KUKA KRL program: EPS_2_251491_MH03_A_20251118025954.src

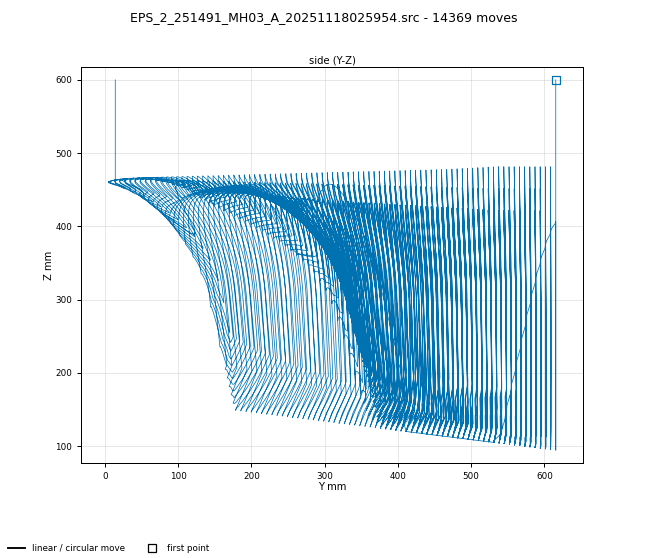
[picture p0: tool path of EPS_2_251491_MH03_A_20251118025954.src, 14369 of 14371 moves have a stored position in this frame; points joined in program order, loops and branches not executed]
&ACCESS RVP
&REL 4
&COMMENT QRS 19112012
&PARAM EDITMASK = *
DEF PART()
EXT BAS (BAS_COMMAND :IN,REAL :IN )
INT I
BAS (#INITMOV,0 )

;KUKA QRS Post kuka4.cps  Date:22-06-2017 !

File_ID=2921

QRS_PRE_INIT()

;Init var - Until changes are made in qrs_pre_init
Outlet_Square_prg=0
Inlet_1_Square_prg=0
Inlet_2_Square_prg=0
Inlet_3_Square_prg=0
Inlet_4_Square_prg=0
Inlet_5_Square_prg=0

Outlet_1={X 0.000, Y 534.640, Z 332.000, B 0.000, E1 0.000 }
Inlet_1={X 0.000, Y 539.010, Z 272.000, B 0.000, E1 90.000 }
Inlet_2={X 0.000, Y 536.830, Z 302.000, B 0.000, E1 207.000 }
Inlet_3={X 0.000, Y 539.010, Z 272.000, B 0.000, E1 270.000 }
Outlet_1_type=299
Inlet_1_type=299
Inlet_2_type=299
Inlet_3_type=299
;QRS#1=Sidecore dimensions
;QRS#2=300-12" PVC SDR 35
;QRS#3=300-12" PVC SDR 35
;QRS#4=300-12" PVC SDR 35
;QRS#5=300-12" PVC SDR 35
;QRS#6=
;QRS#7=
;QRS#8=
;QRS#9=16M PSX
;QRS#10=16M PSX
;QRS#11=16M PSX
;QRS#12=16M PSX
;QRS#13=
;QRS#14=
;QRS#15=
;QRS#16=1220x127x762 2,5'
;QRS#17=EPS Height
;QRS#18=481,5
;QRS#19=*
;QRS#20= UPDATED VERSION 22-06-2017
;QRS#21=*
Outlet_Square=0150
Inlet_1_Square=0150
Inlet_2_Square=0150
Inlet_3_Square=0150
Inlet_4_Square=0
Inlet_5_Square=0
Mill_Square=1
Outlet_Square_Prg=206
Inlet_1_Square_prg=206
Inlet_2_Square_prg=206
Inlet_3_Square_prg=206

QRS_INIT()

$ADVANCE=5

; T1
PTP {E1 173.529,E2 173.529}
PTP {X 0,Y 615.494,A -85,B 0,C 180,E1 173.529,E2 173.529,E3 0,E4 0,E5 0,E6 0}
QRS_SPEED_INIT()
LIN {X 0,Y 615.494,Z 600,A -85,B 0,C 180,E1 173.529,E2 173.529,E3 0,E4 0,E5 0,E6 0} C_VEL
LIN {X 0,Y 615.494,Z 417.846,A -85,B 0,C 180,E1 173.529,E2 173.529} C_VEL
LIN {X 0,Y 615.494,Z 408.199,A -85,B 0,C 180,E1 173.529,E2 173.529} C_VEL
LIN {X 0,Y 615.491,Z 406.378,A -85,B 0,C 180,E1 173.42,E2 173.42} C_VEL
LIN {X 0,Y 615.494,Z 399.659,A -85,B 0,C 180,E1 172.124,E2 172.124} C_VEL
LIN {X 0,Y 615.491,Z 391.142,A -85,B 0,C 180,E1 170.801,E2 170.801} C_VEL
LIN {X 0,Y 615.494,Z 382.064,A -85,B 0,C 180,E1 169.639,E2 169.639} C_VEL
LIN {X 0,Y 615.493,Z 372.79,A -85,B 0,C 180,E1 168.64,E2 168.64} C_VEL
LIN {X 0,Y 615.496,Z 360.819,A -85,B 0,C 180,E1 167.554,E2 167.554} C_VEL
LIN {X 0,Y 615.497,Z 348.577,A -85,B 0,C 180,E1 166.631,E2 166.631} C_VEL
LIN {X 0,Y 615.496,Z 335.878,A -85,B 0,C 180,E1 165.834,E2 165.834} C_VEL
LIN {X 0,Y 615.481,Z 321.775,A -85,B 0,C 180,E1 165.112,E2 165.112} C_VEL
LIN {X 0,Y 615.491,Z 307.115,A -85,B 0,C 180,E1 164.519,E2 164.519} C_VEL
LIN {X 0,Y 615.495,Z 292.173,A -85,B 0,C 180,E1 164.062,E2 164.062} C_VEL
LIN {X 0,Y 615.483,Z 277.013,A -85,B 0,C 180,E1 163.738,E2 163.738} C_VEL
LIN {X 0,Y 615.449,Z 230.182,A -85,B 0,C 180,E1 163.156,E2 163.156} C_VEL
LIN {X 0,Y 615.473,Z 111.41,A -85,B 0,C 180,E1 161.725,E2 161.725} C_VEL
LIN {X 0,Y 615.445,Z 94.319,A -85,B 0,C 180,E1 159.337,E2 159.337} C_VEL
LIN {X 0,Y 615.446,Z 94.317,A -85,B 0,C 180,E1 157.154,E2 157.154} C_VEL
LIN {X 0,Y 615.497,Z 94.322,A -85,B 0,C 180,E1 154.284,E2 154.284} C_VEL
LIN {X 0,Y 615.441,Z 94.32,A -85,B 0,C 180,E1 151.558,E2 151.558} C_VEL
LIN {X 0,Y 615.472,Z 94.315,A -85,B 0,C 180,E1 148.917,E2 148.917} C_VEL
LIN {X 0,Y 615.455,Z 94.322,A -85,B 0,C 180,E1 145.976,E2 145.976} C_VEL
LIN {X 0,Y 615.438,Z 94.319,A -85,B 0,C 180,E1 143.571,E2 143.571} C_VEL
LIN {X 0,Y 615.491,Z 94.314,A -85,B 0,C 180,E1 140.938,E2 140.938} C_VEL
LIN {X 0,Y 615.491,Z 94.325,A -85,B 0,C 180,E1 138.526,E2 138.526} C_VEL
LIN {X 0,Y 615.437,Z 94.32,A -85,B 0,C 180,E1 135.845,E2 135.845} C_VEL
LIN {X 0,Y 615.473,Z 94.316,A -85,B 0,C 180,E1 133.246,E2 133.246} C_VEL
LIN {X 0,Y 615.47,Z 94.325,A -85,B 0,C 180,E1 130.608,E2 130.608} C_VEL
LIN {X 0,Y 615.434,Z 94.321,A -85,B 0,C 180,E1 128.072,E2 128.072} C_VEL
LIN {X 0,Y 615.449,Z 94.319,A -85,B 0,C 180,E1 125.618,E2 125.618} C_VEL
LIN {X 0,Y 615.488,Z 94.319,A -85,B 0,C 180,E1 123.236,E2 123.236} C_VEL
LIN {X 0,Y 615.475,Z 94.326,A -85,B 0,C 180,E1 120.92,E2 120.92} C_VEL
LIN {X 0,Y 615.434,Z 94.322,A -85,B 0,C 180,E1 118.44,E2 118.44} C_VEL
LIN {X 0,Y 615.434,Z 94.322,A -85,B 0,C 180,E1 116.447,E2 116.447} C_VEL
LIN {X 0,Y 615.442,Z 94.319,A -85,B 0,C 180,E1 113.998,E2 113.998} C_VEL
LIN {X 0,Y 615.498,Z 94.321,A -85,B 0,C 180,E1 111.432,E2 111.432} C_VEL
LIN {X 0,Y 615.43,Z 94.322,A -85,B 0,C 180,E1 108.588,E2 108.588} C_VEL
LIN {X 0,Y 615.43,Z 94.321,A -85,B 0,C 180,E1 106.411,E2 106.411} C_VEL
LIN {X 0,Y 615.474,Z 94.319,A -85,B 0,C 180,E1 103.874,E2 103.874} C_VEL
LIN {X 0,Y 615.452,Z 94.324,A -85,B 0,C 180,E1 101.194,E2 101.194} C_VEL
LIN {X 0,Y 615.448,Z 94.324,A -85,B 0,C 180,E1 99.199,E2 99.199} C_VEL
LIN {X 0,Y 615.444,Z 94.324,A -85,B 0,C 180,E1 97.216,E2 97.216} C_VEL
LIN {X 0,Y 615.442,Z 94.324,A -85,B 0,C 180,E1 95.242,E2 95.242} C_VEL
LIN {X 0,Y 615.439,Z 94.324,A -85,B 0,C 180,E1 93.273,E2 93.273} C_VEL
LIN {X 0,Y 615.439,Z 94.324,A -85,B 0,C 180,E1 91.309,E2 91.309} C_VEL
LIN {X 0,Y 615.437,Z 94.324,A -85,B 0,C 180,E1 89.346,E2 89.346} C_VEL
LIN {X 0,Y 615.422,Z 94.323,A -85,B 0,C 180,E1 87.054,E2 87.054} C_VEL
LIN {X 0,Y 615.429,Z 94.45,A -85,B 0,C 180,E1 86.727,E2 86.727} C_VEL
LIN {X 0,Y 615.496,Z 116.011,A -85,B 0,C 180,E1 84.102,E2 84.102} C_VEL
LIN {X 0,Y 615.457,Z 139.488,A -85,B 0,C 180,E1 81.297,E2 81.297} C_VEL
LIN {X 0,Y 615.461,Z 140.359,A -85,B 0,C 180,E1 81.194,E2 81.194} C_VEL
LIN {X 0,Y 615.483,Z 306.431,A -85,B 0,C 180,E1 79.183,E2 79.183} C_VEL
LIN {X 0,Y 615.49,Z 322.253,A -85,B 0,C 180,E1 78.846,E2 78.846} C_VEL
LIN {X 0,Y 615.492,Z 337.135,A -85,B 0,C 180,E1 78.39,E2 78.39} C_VEL
LIN {X 0,Y 615.484,Z 351.621,A -85,B 0,C 180,E1 77.805,E2 77.805} C_VEL
LIN {X 0,Y 615.492,Z 364.804,A -85,B 0,C 180,E1 77.135,E2 77.135} C_VEL
LIN {X 0,Y 615.497,Z 378.348,A -85,B 0,C 180,E1 76.294,E2 76.294} C_VEL
LIN {X 0,Y 615.496,Z 390.691,A -85,B 0,C 180,E1 75.367,E2 75.367} C_VEL
LIN {X 0,Y 615.498,Z 402.836,A -85,B 0,C 180,E1 74.265,E2 74.265} C_VEL
LIN {X 0,Y 615.494,Z 412.304,A -85,B 0,C 180,E1 73.243,E2 73.243} C_VEL
LIN {X 0,Y 615.494,Z 421.614,A -85,B 0,C 180,E1 72.043,E2 72.043} C_VEL
LIN {X 0,Y 615.499,Z 429.36,A -85,B 0,C 180,E1 70.836,E2 70.836} C_VEL
LIN {X 0,Y 615.492,Z 436.603,A -85,B 0,C 180,E1 69.443,E2 69.443} C_VEL
LIN {X 0,Y 615.489,Z 441.591,A -85,B 0,C 180,E1 68.216,E2 68.216} C_VEL
LIN {X 0,Y 615.491,Z 445.012,A -85,B 0,C 180,E1 67.156,E2 67.156} C_VEL
LIN {X 0,Y 615.491,Z 448.343,A -85,B 0,C 180,E1 65.728,E2 65.728} C_VEL
LIN {X 0,Y 615.497,Z 450.291,A -85,B 0,C 180,E1 64.285,E2 64.285} C_VEL
LIN {X 0,Y 615.497,Z 450.862,A -85,B 0,C 180,E1 62.823,E2 62.823} C_VEL
LIN {X 0,Y 615.489,Z 450.009,A -85,B 0,C 180,E1 61.342,E2 61.342} C_VEL
LIN {X 0,Y 615.499,Z 447.661,A -85,B 0,C 180,E1 59.84,E2 59.84} C_VEL
LIN {X 0,Y 615.494,Z 445.438,A -85,B 0,C 180,E1 58.914,E2 58.914} C_VEL
LIN {X 0,Y 615.493,Z 441.026,A -85,B 0,C 180,E1 57.543,E2 57.543} C_VEL
LIN {X 0,Y 615.494,Z 435.413,A -85,B 0,C 180,E1 56.222,E2 56.222} C_VEL
LIN {X 0,Y 615.495,Z 428.822,A -85,B 0,C 180,E1 54.986,E2 54.986} C_VEL
LIN {X 0,Y 615.496,Z 420.566,A -85,B 0,C 180,E1 53.724,E2 53.724} C_VEL
LIN {X 0,Y 615.493,Z 411.416,A -85,B 0,C 180,E1 52.566,E2 52.566} C_VEL
LIN {X 0,Y 615.495,Z 400.419,A -85,B 0,C 180,E1 51.411,E2 51.411} C_VEL
LIN {X 0,Y 615.498,Z 389.171,A -85,B 0,C 180,E1 50.423,E2 50.423} C_VEL
LIN {X 0,Y 615.498,Z 376.955,A -85,B 0,C 180,E1 49.524,E2 49.524} C_VEL
LIN {X 0,Y 615.486,Z 363.705,A -85,B 0,C 180,E1 48.716,E2 48.716} C_VEL
LIN {X 0,Y 615.485,Z 350.829,A -85,B 0,C 180,E1 48.071,E2 48.071} C_VEL
LIN {X 0,Y 615.481,Z 337.051,A -85,B 0,C 180,E1 47.517,E2 47.517} C_VEL
LIN {X 0,Y 615.491,Z 322.944,A -85,B 0,C 180,E1 47.084,E2 47.084} C_VEL
LIN {X 0,Y 615.487,Z 307.916,A -85,B 0,C 180,E1 46.755,E2 46.755} C_VEL
LIN {X 0,Y 615.463,Z 282.895,A -85,B 0,C 180,E1 46.427,E2 46.427} C_VEL
LIN {X 0,Y 615.482,Z 138.564,A -85,B 0,C 180,E1 44.687,E2 44.687} C_VEL
LIN {X 0,Y 615.459,Z 109.066,A -85,B 0,C 180,E1 41.926,E2 41.926} C_VEL
LIN {X 0,Y 615.45,Z 94.318,A -85,B 0,C 180,E1 40.511,E2 40.511} C_VEL
LIN {X 0,Y 615.471,Z 94.322,A -85,B 0,C 180,E1 38.01,E2 38.01} C_VEL
LIN {X 0,Y 615.491,Z 94.319,A -85,B 0,C 180,E1 35.616,E2 35.616} C_VEL
LIN {X 0,Y 615.487,Z 94.31,A -85,B 0,C 180,E1 33.237,E2 33.237} C_VEL
LIN {X 0,Y 615.476,Z 94.314,A -85,B 0,C 180,E1 30.921,E2 30.921} C_VEL
LIN {X 0,Y 615.495,Z 94.324,A -85,B 0,C 180,E1 28.451,E2 28.451} C_VEL
LIN {X 0,Y 615.484,Z 94.31,A -85,B 0,C 180,E1 25.568,E2 25.568} C_VEL
LIN {X 0,Y 615.491,Z 94.325,A -85,B 0,C 180,E1 22.845,E2 22.845} C_VEL
LIN {X 0,Y 615.467,Z 94.321,A -85,B 0,C 180,E1 20.552,E2 20.552} C_VEL
LIN {X 0,Y 615.466,Z 94.35,A -85,B 0,C 180,E1 19.882,E2 19.882} C_VEL
LIN {X 0,Y 615.453,Z 109.792,A -85,B 0,C 180,E1 18.197,E2 18.197} C_VEL
LIN {X 0,Y 615.479,Z 275.634,A -85,B 0,C 180,E1 16.195,E2 16.195} C_VEL
LIN {X 0,Y 615.497,Z 291.607,A -85,B 0,C 180,E1 15.863,E2 15.863} C_VEL
LIN {X 0,Y 615.488,Z 306.971,A -85,B 0,C 180,E1 15.396,E2 15.396} C_VEL
LIN {X 0,Y 615.483,Z 321.657,A -85,B 0,C 180,E1 14.803,E2 14.803} C_VEL
LIN {X 0,Y 615.492,Z 335.629,A -85,B 0,C 180,E1 14.09,E2 14.09} C_VEL
LIN {X 0,Y 615.498,Z 348.487,A -85,B 0,C 180,E1 13.285,E2 13.285} C_VEL
LIN {X 0,Y 615.496,Z 360.741,A -85,B 0,C 180,E1 12.363,E2 12.363} C_VEL
LIN {X 0,Y 615.498,Z 371.895,A -85,B 0,C 180,E1 11.36,E2 11.36} C_VEL
LIN {X 0,Y 615.497,Z 382.701,A -85,B 0,C 180,E1 10.194,E2 10.194} C_VEL
LIN {X 0,Y 615.495,Z 391.683,A -85,B 0,C 180,E1 9.033,E2 9.033} C_VEL
LIN {X 0,Y 615.493,Z 399.117,A -85,B 0,C 180,E1 7.876,E2 7.876} C_VEL
LIN {X 0,Y 615.492,Z 406.051,A -85,B 0,C 180,E1 6.557,E2 6.557} C_VEL
LIN {X 0,Y 615.489,Z 411.497,A -85,B 0,C 180,E1 5.241,E2 5.241} C_VEL
LIN {X 0,Y 615.495,Z 415.619,A -85,B 0,C 180,E1 3.929,E2 3.929} C_VEL
LIN {X 0,Y 615.493,Z 418.525,A -85,B 0,C 180,E1 2.618,E2 2.618} C_VEL
LIN {X 0,Y 615.491,Z 420.276,A -85,B 0,C 180,E1 1.309,E2 1.309} C_VEL
LIN {X 0,Y 615.492,Z 420.884,A -85,B 0,C 180,E1 0,E2 0} C_VEL
LIN {X 0,Y 615.493,Z 420.338,A -85,B 0,C 180,E1 -1.308,E2 -1.308} C_VEL
LIN {X 0,Y 615.496,Z 418.675,A -85,B 0,C 180,E1 -2.618,E2 -2.618} C_VEL
LIN {X 0,Y 615.494,Z 415.862,A -85,B 0,C 180,E1 -3.928,E2 -3.928} C_VEL
LIN {X 0,Y 615.489,Z 411.836,A -85,B 0,C 180,E1 -5.241,E2 -5.241} C_VEL
LIN {X 0,Y 615.491,Z 406.378,A -85,B 0,C 180,E1 -6.58,E2 -6.58} C_VEL
LIN {X 0,Y 615.494,Z 399.662,A -85,B 0,C 180,E1 -7.875,E2 -7.875} C_VEL
LIN {X 0,Y 615.491,Z 391.145,A -85,B 0,C 180,E1 -9.199,E2 -9.199} C_VEL
LIN {X 0,Y 615.494,Z 382.068,A -85,B 0,C 180,E1 -10.36,E2 -10.36} C_VEL
LIN {X 0,Y 615.493,Z 372.794,A -85,B 0,C 180,E1 -11.36,E2 -11.36} C_VEL
LIN {X 0,Y 615.496,Z 360.824,A -85,B 0,C 180,E1 -12.446,E2 -12.446} C_VEL
LIN {X 0,Y 615.497,Z 348.584,A -85,B 0,C 180,E1 -13.369,E2 -13.369} C_VEL
LIN {X 0,Y 615.496,Z 335.881,A -85,B 0,C 180,E1 -14.165,E2 -14.165} C_VEL
LIN {X 0,Y 615.481,Z 321.785,A -85,B 0,C 180,E1 -14.887,E2 -14.887} C_VEL
LIN {X 0,Y 615.491,Z 307.126,A -85,B 0,C 180,E1 -15.48,E2 -15.48} C_VEL
LIN {X 0,Y 615.495,Z 292.187,A -85,B 0,C 180,E1 -15.937,E2 -15.937} C_VEL
LIN {X 0,Y 615.483,Z 277.021,A -85,B 0,C 180,E1 -16.262,E2 -16.262} C_VEL
LIN {X 0,Y 615.449,Z 230.218,A -85,B 0,C 180,E1 -16.844,E2 -16.844} C_VEL
LIN {X 0,Y 615.473,Z 111.412,A -85,B 0,C 180,E1 -18.275,E2 -18.275} C_VEL
LIN {X 0,Y 615.445,Z 94.319,A -85,B 0,C 180,E1 -20.663,E2 -20.663} C_VEL
LIN {X 0,Y 615.445,Z 94.318,A -85,B 0,C 180,E1 -22.846,E2 -22.846} C_VEL
LIN {X 0,Y 615.498,Z 94.322,A -85,B 0,C 180,E1 -25.715,E2 -25.715} C_VEL
LIN {X 0,Y 615.441,Z 94.32,A -85,B 0,C 180,E1 -28.442,E2 -28.442} C_VEL
LIN {X 0,Y 615.472,Z 94.316,A -85,B 0,C 180,E1 -31.083,E2 -31.083} C_VEL
LIN {X 0,Y 615.449,Z 94.322,A -85,B 0,C 180,E1 -34.024,E2 -34.024} C_VEL
LIN {X 0,Y 615.436,Z 94.32,A -85,B 0,C 180,E1 -36.428,E2 -36.428} C_VEL
LIN {X 0,Y 615.49,Z 94.316,A -85,B 0,C 180,E1 -39.062,E2 -39.062} C_VEL
LIN {X 0,Y 615.476,Z 94.325,A -85,B 0,C 180,E1 -41.475,E2 -41.475} C_VEL
LIN {X 0,Y 615.433,Z 94.322,A -85,B 0,C 180,E1 -43.992,E2 -43.992} C_VEL
LIN {X 0,Y 615.43,Z 94.322,A -85,B 0,C 180,E1 -46.008,E2 -46.008} C_VEL
LIN {X 0,Y 615.451,Z 94.32,A -85,B 0,C 180,E1 -48.523,E2 -48.523} C_VEL
LIN {X 0,Y 615.492,Z 94.325,A -85,B 0,C 180,E1 -51.096,E2 -51.096} C_VEL
LIN {X 0,Y 615.432,Z 94.324,A -85,B 0,C 180,E1 -53.571,E2 -53.571} C_VEL
LIN {X 0,Y 615.425,Z 94.322,A -85,B 0,C 180,E1 -55.974,E2 -55.974} C_VEL
LIN {X 0,Y 615.446,Z 94.322,A -85,B 0,C 180,E1 -58.312,E2 -58.312} C_VEL
LIN {X 0,Y 615.479,Z 94.324,A -85,B 0,C 180,E1 -60.593,E2 -60.593} C_VEL
LIN {X 0,Y 615.419,Z 94.324,A -85,B 0,C 180,E1 -63.553,E2 -63.553} C_VEL
LIN {X 0,Y 615.421,Z 94.362,A -85,B 0,C 180,E1 -63.781,E2 -63.781} C_VEL
LIN {X 0,Y 615.485,Z 117.882,A -85,B 0,C 180,E1 -66.331,E2 -66.331} C_VEL
LIN {X 0,Y 615.49,Z 143.927,A -85,B 0,C 180,E1 -69.094,E2 -69.094} C_VEL
LIN {X 0,Y 615.491,Z 169.317,A -85,B 0,C 180,E1 -71.741,E2 -71.741} C_VEL
LIN {X 0,Y 615.483,Z 336.238,A -85,B 0,C 180,E1 -73.769,E2 -73.769} C_VEL
LIN {X 0,Y 615.496,Z 351.712,A -85,B 0,C 180,E1 -74.095,E2 -74.095} C_VEL
LIN {X 0,Y 615.489,Z 367.05,A -85,B 0,C 180,E1 -74.562,E2 -74.562} C_VEL
LIN {X 0,Y 615.484,Z 380.753,A -85,B 0,C 180,E1 -75.113,E2 -75.113} C_VEL
LIN {X 0,Y 615.493,Z 395.046,A -85,B 0,C 180,E1 -75.833,E2 -75.833} C_VEL
LIN {X 0,Y 615.497,Z 407.898,A -85,B 0,C 180,E1 -76.631,E2 -76.631} C_VEL
LIN {X 0,Y 615.495,Z 420.255,A -85,B 0,C 180,E1 -77.554,E2 -77.554} C_VEL
LIN {X 0,Y 615.496,Z 430.606,A -85,B 0,C 180,E1 -78.473,E2 -78.473} C_VEL
LIN {X 0,Y 615.494,Z 440.184,A -85,B 0,C 180,E1 -79.473,E2 -79.473} C_VEL
LIN {X 0,Y 615.494,Z 449.577,A -85,B 0,C 180,E1 -80.636,E2 -80.636} C_VEL
LIN {X 0,Y 615.494,Z 457.381,A -85,B 0,C 180,E1 -81.794,E2 -81.794} C_VEL
LIN {X 0,Y 615.494,Z 464.609,A -85,B 0,C 180,E1 -83.102,E2 -83.102} C_VEL
LIN {X 0,Y 615.499,Z 470.437,A -85,B 0,C 180,E1 -84.43,E2 -84.43} C_VEL
LIN {X 0,Y 615.491,Z 473.86,A -85,B 0,C 180,E1 -85.415,E2 -85.415} C_VEL
LIN {X 0,Y 615.493,Z 477.318,A -85,B 0,C 180,E1 -86.727,E2 -86.727} C_VEL
LIN {X 0,Y 615.5,Z 479.593,A -85,B 0,C 180,E1 -88.037,E2 -88.037} C_VEL
LIN {X 0,Y 615.491,Z 480.741,A -85,B 0,C 180,E1 -89.346,E2 -89.346} C_VEL
LIN {X 0,Y 615.491,Z 480.741,A -85,B 0,C 180,E1 -90.654,E2 -90.654} C_VEL
LIN {X 0,Y 615.5,Z 479.593,A -85,B 0,C 180,E1 -91.963,E2 -91.963} C_VEL
LIN {X 0,Y 615.493,Z 477.318,A -85,B 0,C 180,E1 -93.273,E2 -93.273} C_VEL
LIN {X 0,Y 615.491,Z 473.86,A -85,B 0,C 180,E1 -94.585,E2 -94.585} C_VEL
LIN {X 0,Y 615.499,Z 469.142,A -85,B 0,C 180,E1 -95.898,E2 -95.898} C_VEL
LIN {X 0,Y 615.492,Z 463.03,A -85,B 0,C 180,E1 -97.216,E2 -97.216} C_VEL
LIN {X 0,Y 615.493,Z 455.332,A -85,B 0,C 180,E1 -98.537,E2 -98.537} C_VEL
LIN {X 0,Y 615.495,Z 447.113,A -85,B 0,C 180,E1 -99.696,E2 -99.696} C_VEL
LIN {X 0,Y 615.496,Z 436.899,A -85,B 0,C 180,E1 -100.892,E2 -100.892} C_VEL
LIN {X 0,Y 615.496,Z 427.067,A -85,B 0,C 180,E1 -101.861,E2 -101.861} C_VEL
LIN {X 0,Y 615.497,Z 414.947,A -85,B 0,C 180,E1 -102.865,E2 -102.865} C_VEL
LIN {X 0,Y 615.498,Z 402.797,A -85,B 0,C 180,E1 -103.706,E2 -103.706} C_VEL
LIN {X 0,Y 615.477,Z 389.379,A -85,B 0,C 180,E1 -104.473,E2 -104.473} C_VEL
LIN {X 0,Y 615.497,Z 374.847,A -85,B 0,C 180,E1 -105.141,E2 -105.141} C_VEL
LIN {X 0,Y 615.494,Z 360.614,A -85,B 0,C 180,E1 -105.65,E2 -105.65} C_VEL
LIN {X 0,Y 615.498,Z 346.199,A -85,B 0,C 180,E1 -106.034,E2 -106.034} C_VEL
LIN {X 0,Y 615.474,Z 331.9,A -85,B 0,C 180,E1 -106.293,E2 -106.293} C_VEL
LIN {X 0,Y 615.454,Z 167.704,A -85,B 0,C 180,E1 -108.274,E2 -108.274} C_VEL
LIN {X 0,Y 615.424,Z 138.767,A -85,B 0,C 180,E1 -110.637,E2 -110.637} C_VEL
LIN {X 0,Y 615.499,Z 105.726,A -85,B 0,C 180,E1 -113.378,E2 -113.378} C_VEL
LIN {X 0,Y 615.426,Z 94.322,A -85,B 0,C 180,E1 -114.364,E2 -114.364} C_VEL
LIN {X 0,Y 615.475,Z 94.324,A -85,B 0,C 180,E1 -117.043,E2 -117.043} C_VEL
LIN {X 0,Y 615.446,Z 94.32,A -85,B 0,C 180,E1 -119.788,E2 -119.788} C_VEL
LIN {X 0,Y 615.43,Z 94.322,A -85,B 0,C 180,E1 -122.322,E2 -122.322} C_VEL
LIN {X 0,Y 615.471,Z 94.324,A -85,B 0,C 180,E1 -124.816,E2 -124.816} C_VEL
LIN {X 0,Y 615.487,Z 94.318,A -85,B 0,C 180,E1 -127.242,E2 -127.242} C_VEL
LIN {X 0,Y 615.434,Z 94.32,A -85,B 0,C 180,E1 -129.754,E2 -129.754} C_VEL
LIN {X 0,Y 615.432,Z 94.322,A -85,B 0,C 180,E1 -132.075,E2 -132.075} C_VEL
LIN {X 0,Y 615.437,Z 94.322,A -85,B 0,C 180,E1 -134.154,E2 -134.154} C_VEL
LIN {X 0,Y 615.488,Z 94.319,A -85,B 0,C 180,E1 -136.953,E2 -136.953} C_VEL
LIN {X 0,Y 615.446,Z 94.319,A -85,B 0,C 180,E1 -139.39,E2 -139.39} C_VEL
LIN {X 0,Y 615.435,Z 94.322,A -85,B 0,C 180,E1 -141.928,E2 -141.928} C_VEL
LIN {X 0,Y 615.481,Z 94.324,A -85,B 0,C 180,E1 -144.384,E2 -144.384} C_VEL
LIN {X 0,Y 615.486,Z 94.318,A -85,B 0,C 180,E1 -146.764,E2 -146.764} C_VEL
LIN {X 0,Y 615.454,Z 94.317,A -85,B 0,C 180,E1 -149.079,E2 -149.079} C_VEL
LIN {X 0,Y 615.436,Z 94.32,A -85,B 0,C 180,E1 -151.559,E2 -151.559} C_VEL
LIN {X 0,Y 615.494,Z 94.32,A -85,B 0,C 180,E1 -154.43,E2 -154.43} C_VEL
LIN {X 0,Y 615.439,Z 94.319,A -85,B 0,C 180,E1 -157.154,E2 -157.154} C_VEL
LIN {X 0,Y 615.439,Z 94.35,A -85,B 0,C 180,E1 -159.432,E2 -159.432} C_VEL
LIN {X 0,Y 615.467,Z 111.616,A -85,B 0,C 180,E1 -161.825,E2 -161.825} C_VEL
LIN {X 0,Y 615.478,Z 275.687,A -85,B 0,C 180,E1 -163.805,E2 -163.805} C_VEL
LIN {X 0,Y 615.497,Z 291.624,A -85,B 0,C 180,E1 -164.138,E2 -164.138} C_VEL
LIN {X 0,Y 615.488,Z 306.982,A -85,B 0,C 180,E1 -164.605,E2 -164.605} C_VEL
LIN {X 0,Y 615.483,Z 321.666,A -85,B 0,C 180,E1 -165.197,E2 -165.197} C_VEL
LIN {X 0,Y 615.492,Z 335.63,A -85,B 0,C 180,E1 -165.91,E2 -165.91} C_VEL
LIN {X 0,Y 615.498,Z 348.494,A -85,B 0,C 180,E1 -166.715,E2 -166.715} C_VEL
LIN {X 0,Y 615.496,Z 360.746,A -85,B 0,C 180,E1 -167.638,E2 -167.638} C_VEL
LIN {X 0,Y 615.498,Z 371.9,A -85,B 0,C 180,E1 -168.641,E2 -168.641} C_VEL
LIN {X 0,Y 615.497,Z 382.704,A -85,B 0,C 180,E1 -169.806,E2 -169.806} C_VEL
LIN {X 0,Y 615.495,Z 391.686,A -85,B 0,C 180,E1 -170.967,E2 -170.967} C_VEL
LIN {X 0,Y 615.493,Z 399.12,A -85,B 0,C 180,E1 -172.125,E2 -172.125} C_VEL
LIN {X 0,Y 615.492,Z 406.053,A -85,B 0,C 180,E1 -173.444,E2 -173.444} C_VEL
LIN {X 0,Y 615.489,Z 411.499,A -85,B 0,C 180,E1 -174.759,E2 -174.759} C_VEL
LIN {X 0,Y 615.495,Z 415.62,A -85,B 0,C 180,E1 -176.072,E2 -176.072} C_VEL
LIN {X 0,Y 615.493,Z 418.526,A -85,B 0,C 180,E1 -177.382,E2 -177.382} C_VEL
LIN {X 0,Y 615.491,Z 420.276,A -85,B 0,C 180,E1 -178.692,E2 -178.692} C_VEL
LIN {X 0,Y 615.492,Z 420.885,A -85,B 0,C 180,E1 -180,E2 -180} C_VEL
LIN {X 0,Y 615.493,Z 420.338,A -85,B 0,C 180,E1 -181.309,E2 -181.309} C_VEL
LIN {X 0,Y 615.496,Z 418.674,A -85,B 0,C 180,E1 -182.618,E2 -182.618} C_VEL
LIN {X 0,Y 615.494,Z 415.86,A -85,B 0,C 180,E1 -183.929,E2 -183.929} C_VEL
LIN {X 0,Y 615.489,Z 411.834,A -85,B 0,C 180,E1 -185.241,E2 -185.241} C_VEL
LIN {X 0,Y 615.491,Z 406.378,A -85,B 0,C 180,E1 -186.58,E2 -186.58} C_VEL
LIN {X 0,Y 614.829,Z 404.12,A -85,B 0,C 180,E1 -187.078,E2 -187.078} C_VEL
LIN {X 0,Y 612.01,Z 400.228,A -85,B 0,C 180,E1 -187.885,E2 -187.885} C_VEL
LIN {X 0,Y 609.156,Z 395.66,A -85,B 0,C 180,E1 -188.676,E2 -188.676} C_VEL
LIN {X 0,Y 608.465,Z 392.513,A -85,B 0,C 180,E1 -189.149,E2 -189.149} C_VEL
LIN {X 0,Y 608.476,Z 383.663,A -85,B 0,C 180,E1 -190.313,E2 -190.313} C_VEL
LIN {X 0,Y 608.495,Z 372.944,A -85,B 0,C 180,E1 -191.492,E2 -191.492} C_VEL
LIN {X 0,Y 608.513,Z 360.9,A -85,B 0,C 180,E1 -192.592,E2 -192.592} C_VEL
LIN {X 0,Y 608.543,Z 348.613,A -85,B 0,C 180,E1 -193.525,E2 -193.525} C_VEL
LIN {X 0,Y 608.585,Z 335.656,A -85,B 0,C 180,E1 -194.342,E2 -194.342} C_VEL
LIN {X 0,Y 608.584,Z 321.764,A -85,B 0,C 180,E1 -195.06,E2 -195.06} C_VEL
LIN {X 0,Y 608.645,Z 307.074,A -85,B 0,C 180,E1 -195.659,E2 -195.659} C_VEL
LIN {X 0,Y 608.661,Z 291.541,A -85,B 0,C 180,E1 -196.138,E2 -196.138} C_VEL
LIN {X 0,Y 608.674,Z 275.81,A -85,B 0,C 180,E1 -196.469,E2 -196.469} C_VEL
LIN {X 0,Y 608.632,Z 112.332,A -85,B 0,C 180,E1 -198.468,E2 -198.468} C_VEL
LIN {X 0,Y 608.502,Z 111.442,A -85,B 0,C 180,E1 -198.492,E2 -198.492} C_VEL
LIN {X 0,Y 608.459,Z 95.565,A -85,B 0,C 180,E1 -200.734,E2 -200.734} C_VEL
LIN {X 0,Y 608.428,Z 95.317,A -85,B 0,C 180,E1 -200.782,E2 -200.782} C_VEL
LIN {X 0,Y 608.431,Z 95.316,A -85,B 0,C 180,E1 -203.125,E2 -203.125} C_VEL
LIN {X 0,Y 608.433,Z 95.322,A -85,B 0,C 180,E1 -206.036,E2 -206.036} C_VEL
LIN {X 0,Y 608.436,Z 95.315,A -85,B 0,C 180,E1 -208.613,E2 -208.613} C_VEL
LIN {X 0,Y 608.446,Z 95.318,A -85,B 0,C 180,E1 -211.318,E2 -211.318} C_VEL
LIN {X 0,Y 608.448,Z 95.322,A -85,B 0,C 180,E1 -213.731,E2 -213.731} C_VEL
LIN {X 0,Y 608.434,Z 95.317,A -85,B 0,C 180,E1 -216.093,E2 -216.093} C_VEL
LIN {X 0,Y 608.418,Z 95.317,A -85,B 0,C 180,E1 -218.592,E2 -218.592} C_VEL
LIN {X 0,Y 608.466,Z 95.32,A -85,B 0,C 180,E1 -221.342,E2 -221.342} C_VEL
LIN {X 0,Y 608.436,Z 95.317,A -85,B 0,C 180,E1 -223.873,E2 -223.873} C_VEL
LIN {X 0,Y 608.461,Z 95.313,A -85,B 0,C 180,E1 -226.693,E2 -226.693} C_VEL
LIN {X 0,Y 608.436,Z 95.318,A -85,B 0,C 180,E1 -229.673,E2 -229.673} C_VEL
LIN {X 0,Y 608.48,Z 95.315,A -85,B 0,C 180,E1 -232.841,E2 -232.841} C_VEL
LIN {X 0,Y 608.444,Z 95.316,A -85,B 0,C 180,E1 -235.529,E2 -235.529} C_VEL
LIN {X 0,Y 608.426,Z 95.316,A -85,B 0,C 180,E1 -237.903,E2 -237.903} C_VEL
LIN {X 0,Y 608.435,Z 95.316,A -85,B 0,C 180,E1 -240.219,E2 -240.219} C_VEL
LIN {X 0,Y 608.482,Z 95.319,A -85,B 0,C 180,E1 -242.793,E2 -242.793} C_VEL
LIN {X 0,Y 608.422,Z 95.317,A -85,B 0,C 180,E1 -245.428,E2 -245.428} C_VEL
LIN {X 0,Y 608.458,Z 95.316,A -85,B 0,C 180,E1 -248.308,E2 -248.308} C_VEL
LIN {X 0,Y 608.417,Z 95.318,A -85,B 0,C 180,E1 -251.3,E2 -251.3} C_VEL
LIN {X 0,Y 608.428,Z 95.317,A -85,B 0,C 180,E1 -253.905,E2 -253.905} C_VEL
LIN {X 0,Y 608.438,Z 95.322,A -85,B 0,C 180,E1 -256.643,E2 -256.643} C_VEL
LIN {X 0,Y 608.411,Z 95.318,A -85,B 0,C 180,E1 -259.349,E2 -259.349} C_VEL
LIN {X 0,Y 608.469,Z 95.316,A -85,B 0,C 180,E1 -262.033,E2 -262.033} C_VEL
LIN {X 0,Y 608.429,Z 95.319,A -85,B 0,C 180,E1 -264.698,E2 -264.698} C_VEL
LIN {X 0,Y 608.425,Z 95.316,A -85,B 0,C 180,E1 -267.352,E2 -267.352} C_VEL
LIN {X 0,Y 608.476,Z 95.318,A -85,B 0,C 180,E1 -270,E2 -270} C_VEL
LIN {X 0,Y 608.431,Z 95.319,A -85,B 0,C 180,E1 -272.648,E2 -272.648} C_VEL
LIN {X 0,Y 608.421,Z 95.427,A -85,B 0,C 180,E1 -273.104,E2 -273.104} C_VEL
LIN {X 0,Y 608.572,Z 106.424,A -85,B 0,C 180,E1 -274.471,E2 -274.471} C_VEL
LIN {X 0,Y 608.535,Z 126.598,A -85,B 0,C 180,E1 -276.932,E2 -276.932} C_VEL
LIN {X 0,Y 608.514,Z 140.4,A -85,B 0,C 180,E1 -278.593,E2 -278.593} C_VEL
LIN {X 0,Y 608.745,Z 154.874,A -85,B 0,C 180,E1 -278.778,E2 -278.778} C_VEL
LIN {X 0,Y 608.676,Z 306.078,A -85,B 0,C 180,E1 -280.625,E2 -280.625} C_VEL
LIN {X 0,Y 608.667,Z 321.081,A -85,B 0,C 180,E1 -280.942,E2 -280.942} C_VEL
LIN {X 0,Y 608.638,Z 336.36,A -85,B 0,C 180,E1 -281.405,E2 -281.405} C_VEL
LIN {X 0,Y 608.615,Z 351.02,A -85,B 0,C 180,E1 -281.997,E2 -281.997} C_VEL
LIN {X 0,Y 608.558,Z 365.88,A -85,B 0,C 180,E1 -282.76,E2 -282.76} C_VEL
LIN {X 0,Y 608.555,Z 379.258,A -85,B 0,C 180,E1 -283.61,E2 -283.61} C_VEL
LIN {X 0,Y 608.527,Z 391.493,A -85,B 0,C 180,E1 -284.548,E2 -284.548} C_VEL
LIN {X 0,Y 608.505,Z 402.743,A -85,B 0,C 180,E1 -285.577,E2 -285.577} C_VEL
LIN {X 0,Y 608.475,Z 412.225,A -85,B 0,C 180,E1 -286.603,E2 -286.603} C_VEL
LIN {X 0,Y 608.455,Z 421.716,A -85,B 0,C 180,E1 -287.824,E2 -287.824} C_VEL
LIN {X 0,Y 608.465,Z 429.549,A -85,B 0,C 180,E1 -289.044,E2 -289.044} C_VEL
LIN {X 0,Y 608.438,Z 436.038,A -85,B 0,C 180,E1 -290.275,E2 -290.275} C_VEL
LIN {X 0,Y 608.423,Z 441.978,A -85,B 0,C 180,E1 -291.693,E2 -291.693} C_VEL
LIN {X 0,Y 608.431,Z 446.432,A -85,B 0,C 180,E1 -293.125,E2 -293.125} C_VEL
LIN {X 0,Y 608.41,Z 449.478,A -85,B 0,C 180,E1 -294.573,E2 -294.573} C_VEL
LIN {X 0,Y 608.422,Z 451.135,A -85,B 0,C 180,E1 -296.037,E2 -296.037} C_VEL
LIN {X 0,Y 608.427,Z 451.395,A -85,B 0,C 180,E1 -297.519,E2 -297.519} C_VEL
LIN {X 0,Y 608.412,Z 450.2,A -85,B 0,C 180,E1 -299.023,E2 -299.023} C_VEL
LIN {X 0,Y 608.436,Z 448.723,A -85,B 0,C 180,E1 -299.966,E2 -299.966} C_VEL
LIN {X 0,Y 608.423,Z 445.486,A -85,B 0,C 180,E1 -301.319,E2 -301.319} C_VEL
LIN {X 0,Y 608.426,Z 441.532,A -85,B 0,C 180,E1 -302.516,E2 -302.516} C_VEL
LIN {X 0,Y 608.431,Z 436.459,A -85,B 0,C 180,E1 -303.728,E2 -303.728} C_VEL
LIN {X 0,Y 608.465,Z 429.454,A -85,B 0,C 180,E1 -305.061,E2 -305.061} C_VEL
LIN {X 0,Y 608.46,Z 421.496,A -85,B 0,C 180,E1 -306.296,E2 -306.296} C_VEL
LIN {X 0,Y 608.477,Z 412.787,A -85,B 0,C 180,E1 -307.421,E2 -307.421} C_VEL
LIN {X 0,Y 608.49,Z 402.001,A -85,B 0,C 180,E1 -308.586,E2 -308.586} C_VEL
LIN {X 0,Y 608.509,Z 390.162,A -85,B 0,C 180,E1 -309.651,E2 -309.651} C_VEL
LIN {X 0,Y 608.533,Z 378.782,A -85,B 0,C 180,E1 -310.514,E2 -310.514} C_VEL
LIN {X 0,Y 608.565,Z 365.472,A -85,B 0,C 180,E1 -311.353,E2 -311.353} C_VEL
LIN {X 0,Y 608.589,Z 351.953,A -85,B 0,C 180,E1 -312.051,E2 -312.051} C_VEL
LIN {X 0,Y 608.613,Z 336.996,A -85,B 0,C 180,E1 -312.664,E2 -312.664} C_VEL
LIN {X 0,Y 608.659,Z 321.145,A -85,B 0,C 180,E1 -313.147,E2 -313.147} C_VEL
LIN {X 0,Y 608.684,Z 306.247,A -85,B 0,C 180,E1 -313.462,E2 -313.462} C_VEL
LIN {X 0,Y 608.696,Z 139.384,A -85,B 0,C 180,E1 -315.502,E2 -315.502} C_VEL
LIN {X 0,Y 608.594,Z 138.174,A -85,B 0,C 180,E1 -315.564,E2 -315.564} C_VEL
LIN {X 0,Y 608.63,Z 108.852,A -85,B 0,C 180,E1 -318.342,E2 -318.342} C_VEL
LIN {X 0,Y 608.522,Z 95.754,A -85,B 0,C 180,E1 -319.604,E2 -319.604} C_VEL
LIN {X 0,Y 608.419,Z 95.32,A -85,B 0,C 180,E1 -319.694,E2 -319.694} C_VEL
LIN {X 0,Y 608.463,Z 95.322,A -85,B 0,C 180,E1 -322.253,E2 -322.253} C_VEL
LIN {X 0,Y 608.438,Z 95.315,A -85,B 0,C 180,E1 -325.096,E2 -325.096} C_VEL
LIN {X 0,Y 608.453,Z 95.317,A -85,B 0,C 180,E1 -327.479,E2 -327.479} C_VEL
LIN {X 0,Y 608.466,Z 95.314,A -85,B 0,C 180,E1 -330.22,E2 -330.22} C_VEL
LIN {X 0,Y 608.479,Z 95.311,A -85,B 0,C 180,E1 -332.793,E2 -332.793} C_VEL
LIN {X 0,Y 608.447,Z 95.323,A -85,B 0,C 180,E1 -335.428,E2 -335.428} C_VEL
LIN {X 0,Y 608.466,Z 95.312,A -85,B 0,C 180,E1 -338.308,E2 -338.308} C_VEL
LIN {X 0,Y 608.452,Z 95.347,A -85,B 0,C 180,E1 -339.99,E2 -339.99} C_VEL
LIN {X 0,Y 608.518,Z 109.823,A -85,B 0,C 180,E1 -341.588,E2 -341.588} C_VEL
LIN {X 0,Y 608.726,Z 126.388,A -85,B 0,C 180,E1 -341.796,E2 -341.796} C_VEL
LIN {X 0,Y 608.678,Z 275.601,A -85,B 0,C 180,E1 -343.619,E2 -343.619} C_VEL
LIN {X 0,Y 608.666,Z 291.629,A -85,B 0,C 180,E1 -343.955,E2 -343.955} C_VEL
LIN {X 0,Y 608.618,Z 306.96,A -85,B 0,C 180,E1 -344.426,E2 -344.426} C_VEL
LIN {X 0,Y 608.589,Z 321.649,A -85,B 0,C 180,E1 -345.025,E2 -345.025} C_VEL
LIN {X 0,Y 608.562,Z 335.572,A -85,B 0,C 180,E1 -345.742,E2 -345.742} C_VEL
LIN {X 0,Y 608.548,Z 348.543,A -85,B 0,C 180,E1 -346.56,E2 -346.56} C_VEL
LIN {X 0,Y 608.504,Z 360.83,A -85,B 0,C 180,E1 -347.493,E2 -347.493} C_VEL
LIN {X 0,Y 608.498,Z 372.044,A -85,B 0,C 180,E1 -348.508,E2 -348.508} C_VEL
LIN {X 0,Y 608.477,Z 382.929,A -85,B 0,C 180,E1 -349.687,E2 -349.687} C_VEL
LIN {X 0,Y 608.469,Z 391.977,A -85,B 0,C 180,E1 -350.862,E2 -350.862} C_VEL
LIN {X 0,Y 608.456,Z 399.477,A -85,B 0,C 180,E1 -352.033,E2 -352.033} C_VEL
LIN {X 0,Y 608.442,Z 406.643,A -85,B 0,C 180,E1 -353.399,E2 -353.399} C_VEL
LIN {X 0,Y 608.435,Z 411.994,A -85,B 0,C 180,E1 -354.698,E2 -354.698} C_VEL
LIN {X 0,Y 608.432,Z 416.166,A -85,B 0,C 180,E1 -356.026,E2 -356.026} C_VEL
LIN {X 0,Y 608.421,Z 419.11,A -85,B 0,C 180,E1 -357.351,E2 -357.351} C_VEL
LIN {X 0,Y 608.444,Z 420.881,A -85,B 0,C 180,E1 -358.676,E2 -358.676} C_VEL
LIN {X 0,Y 608.432,Z 421.495,A -85,B 0,C 180,E1 -360,E2 -360} C_VEL
LIN {X 0,Y 608.445,Z 420.945,A -85,B 0,C 180,E1 -361.324,E2 -361.324} C_VEL
LIN {X 0,Y 608.424,Z 419.26,A -85,B 0,C 180,E1 -362.648,E2 -362.648} C_VEL
LIN {X 0,Y 608.431,Z 416.408,A -85,B 0,C 180,E1 -363.974,E2 -363.974} C_VEL
LIN {X 0,Y 608.435,Z 412.33,A -85,B 0,C 180,E1 -365.302,E2 -365.302} C_VEL
LIN {X 0,Y 608.445,Z 406.923,A -85,B 0,C 180,E1 -366.633,E2 -366.633} C_VEL
LIN {X 0,Y 608.457,Z 400.021,A -85,B 0,C 180,E1 -367.967,E2 -367.967} C_VEL
LIN {X 0,Y 608.466,Z 392.593,A -85,B 0,C 180,E1 -369.138,E2 -369.138} C_VEL
LIN {X 0,Y 608.476,Z 383.661,A -85,B 0,C 180,E1 -370.313,E2 -370.313} C_VEL
LIN {X 0,Y 608.495,Z 372.951,A -85,B 0,C 180,E1 -371.492,E2 -371.492} C_VEL
LIN {X 0,Y 608.513,Z 360.899,A -85,B 0,C 180,E1 -372.591,E2 -372.591} C_VEL
LIN {X 0,Y 608.543,Z 348.622,A -85,B 0,C 180,E1 -373.525,E2 -373.525} C_VEL
LIN {X 0,Y 608.584,Z 335.678,A -85,B 0,C 180,E1 -374.342,E2 -374.342} C_VEL
LIN {X 0,Y 608.583,Z 321.755,A -85,B 0,C 180,E1 -375.06,E2 -375.06} C_VEL
LIN {X 0,Y 608.645,Z 307.084,A -85,B 0,C 180,E1 -375.659,E2 -375.659} C_VEL
LIN {X 0,Y 608.66,Z 291.561,A -85,B 0,C 180,E1 -376.137,E2 -376.137} C_VEL
LIN {X 0,Y 608.673,Z 275.786,A -85,B 0,C 180,E1 -376.469,E2 -376.469} C_VEL
LIN {X 0,Y 608.632,Z 112.351,A -85,B 0,C 180,E1 -378.468,E2 -378.468} C_VEL
LIN {X 0,Y 608.502,Z 111.444,A -85,B 0,C 180,E1 -378.492,E2 -378.492} C_VEL
LIN {X 0,Y 608.458,Z 95.566,A -85,B 0,C 180,E1 -380.734,E2 -380.734} C_VEL
LIN {X 0,Y 608.427,Z 95.317,A -85,B 0,C 180,E1 -380.781,E2 -380.781} C_VEL
LIN {X 0,Y 608.43,Z 95.316,A -85,B 0,C 180,E1 -383.125,E2 -383.125} C_VEL
LIN {X 0,Y 608.432,Z 95.322,A -85,B 0,C 180,E1 -386.036,E2 -386.036} C_VEL
LIN {X 0,Y 608.435,Z 95.315,A -85,B 0,C 180,E1 -388.613,E2 -388.613} C_VEL
LIN {X 0,Y 608.444,Z 95.319,A -85,B 0,C 180,E1 -391.318,E2 -391.318} C_VEL
LIN {X 0,Y 608.446,Z 95.321,A -85,B 0,C 180,E1 -393.731,E2 -393.731} C_VEL
LIN {X 0,Y 608.431,Z 95.317,A -85,B 0,C 180,E1 -396.093,E2 -396.093} C_VEL
LIN {X 0,Y 608.414,Z 95.318,A -85,B 0,C 180,E1 -398.592,E2 -398.592} C_VEL
LIN {X 0,Y 608.458,Z 95.323,A -85,B 0,C 180,E1 -401.342,E2 -401.342} C_VEL
LIN {X 0,Y 608.43,Z 95.317,A -85,B 0,C 180,E1 -403.873,E2 -403.873} C_VEL
LIN {X 0,Y 608.459,Z 95.315,A -85,B 0,C 180,E1 -406.692,E2 -406.692} C_VEL
LIN {X 0,Y 608.432,Z 95.317,A -85,B 0,C 180,E1 -409.673,E2 -409.673} C_VEL
LIN {X 0,Y 608.477,Z 95.318,A -85,B 0,C 180,E1 -412.841,E2 -412.841} C_VEL
LIN {X 0,Y 608.43,Z 95.317,A -85,B 0,C 180,E1 -415.528,E2 -415.528} C_VEL
LIN {X 0,Y 608.416,Z 95.317,A -85,B 0,C 180,E1 -417.903,E2 -417.903} C_VEL
LIN {X 0,Y 608.428,Z 95.318,A -85,B 0,C 180,E1 -420.218,E2 -420.218} C_VEL
LIN {X 0,Y 608.466,Z 95.321,A -85,B 0,C 180,E1 -422.795,E2 -422.795} C_VEL
LIN {X 0,Y 608.402,Z 95.403,A -85,B 0,C 180,E1 -423.57,E2 -423.57} C_VEL
LIN {X 0,Y 608.691,Z 101.304,A -85,B 0,C 180,E1 -424.236,E2 -424.236} C_VEL
LIN {X 0,Y 608.665,Z 125.6,A -85,B 0,C 180,E1 -426.885,E2 -426.885} C_VEL
LIN {X 0,Y 608.592,Z 152.258,A -85,B 0,C 180,E1 -429.73,E2 -429.73} C_VEL
LIN {X 0,Y 608.574,Z 169.418,A -85,B 0,C 180,E1 -431.536,E2 -431.536} C_VEL
LIN {X 0,Y 608.743,Z 196.998,A -85,B 0,C 180,E1 -431.881,E2 -431.881} C_VEL
LIN {X 0,Y 608.677,Z 336.238,A -85,B 0,C 180,E1 -433.583,E2 -433.583} C_VEL
LIN {X 0,Y 608.671,Z 351.711,A -85,B 0,C 180,E1 -433.912,E2 -433.912} C_VEL
LIN {X 0,Y 608.631,Z 367.048,A -85,B 0,C 180,E1 -434.384,E2 -434.384} C_VEL
LIN {X 0,Y 608.605,Z 380.757,A -85,B 0,C 180,E1 -434.94,E2 -434.94} C_VEL
LIN {X 0,Y 608.572,Z 394.237,A -85,B 0,C 180,E1 -435.624,E2 -435.624} C_VEL
LIN {X 0,Y 608.554,Z 406.664,A -85,B 0,C 180,E1 -436.39,E2 -436.39} C_VEL
LIN {X 0,Y 608.528,Z 419.283,A -85,B 0,C 180,E1 -437.324,E2 -437.324} C_VEL
LIN {X 0,Y 608.497,Z 430.748,A -85,B 0,C 180,E1 -438.339,E2 -438.339} C_VEL
LIN {X 0,Y 608.475,Z 440.388,A -85,B 0,C 180,E1 -439.35,E2 -439.35} C_VEL
LIN {X 0,Y 608.477,Z 449.854,A -85,B 0,C 180,E1 -440.527,E2 -440.527} C_VEL
LIN {X 0,Y 608.456,Z 457.729,A -85,B 0,C 180,E1 -441.699,E2 -441.699} C_VEL
LIN {X 0,Y 608.439,Z 465.087,A -85,B 0,C 180,E1 -443.034,E2 -443.034} C_VEL
LIN {X 0,Y 608.451,Z 470.924,A -85,B 0,C 180,E1 -444.366,E2 -444.366} C_VEL
LIN {X 0,Y 608.427,Z 474.383,A -85,B 0,C 180,E1 -445.362,E2 -445.362} C_VEL
LIN {X 0,Y 608.421,Z 477.886,A -85,B 0,C 180,E1 -446.689,E2 -446.689} C_VEL
LIN {X 0,Y 608.444,Z 480.191,A -85,B 0,C 180,E1 -448.014,E2 -448.014} C_VEL
LIN {X 0,Y 608.434,Z 481.35,A -85,B 0,C 180,E1 -449.338,E2 -449.338} C_VEL
LIN {X 0,Y 608.434,Z 481.35,A -85,B 0,C 180,E1 -450.662,E2 -450.662} C_VEL
LIN {X 0,Y 608.444,Z 480.191,A -85,B 0,C 180,E1 -451.986,E2 -451.986} C_VEL
LIN {X 0,Y 608.421,Z 477.885,A -85,B 0,C 180,E1 -453.311,E2 -453.311} C_VEL
LIN {X 0,Y 608.427,Z 474.383,A -85,B 0,C 180,E1 -454.638,E2 -454.638} C_VEL
LIN {X 0,Y 608.437,Z 469.608,A -85,B 0,C 180,E1 -455.967,E2 -455.967} C_VEL
LIN {X 0,Y 608.456,Z 463.426,A -85,B 0,C 180,E1 -457.3,E2 -457.3} C_VEL
LIN {X 0,Y 608.467,Z 455.654,A -85,B 0,C 180,E1 -458.636,E2 -458.636} C_VEL
LIN {X 0,Y 608.471,Z 447.37,A -85,B 0,C 180,E1 -459.809,E2 -459.809} C_VEL
LIN {X 0,Y 608.492,Z 436.652,A -85,B 0,C 180,E1 -461.063,E2 -461.063} C_VEL
LIN {X 0,Y 608.522,Z 425.274,A -85,B 0,C 180,E1 -462.168,E2 -462.168} C_VEL
LIN {X 0,Y 608.547,Z 413.854,A -85,B 0,C 180,E1 -463.1,E2 -463.1} C_VEL
LIN {X 0,Y 608.563,Z 401.447,A -85,B 0,C 180,E1 -463.95,E2 -463.95} C_VEL
LIN {X 0,Y 608.561,Z 387.859,A -85,B 0,C 180,E1 -464.718,E2 -464.718} C_VEL
LIN {X 0,Y 608.638,Z 373.791,A -85,B 0,C 180,E1 -465.359,E2 -465.359} C_VEL
LIN {X 0,Y 608.644,Z 359.3,A -85,B 0,C 180,E1 -465.874,E2 -465.874} C_VEL
LIN {X 0,Y 608.677,Z 344.108,A -85,B 0,C 180,E1 -466.268,E2 -466.268} C_VEL
LIN {X 0,Y 608.673,Z 328.447,A -85,B 0,C 180,E1 -466.53,E2 -466.53} C_VEL
LIN {X 0,Y 608.644,Z 168.189,A -85,B 0,C 180,E1 -468.473,E2 -468.473} C_VEL
LIN {X 0,Y 608.573,Z 162.041,A -85,B 0,C 180,E1 -468.953,E2 -468.953} C_VEL
LIN {X 0,Y 608.684,Z 129.102,A -85,B 0,C 180,E1 -471.684,E2 -471.684} C_VEL
LIN {X 0,Y 608.702,Z 99.323,A -85,B 0,C 180,E1 -474.2,E2 -474.2} C_VEL
LIN {X 0,Y 608.495,Z 95.848,A -85,B 0,C 180,E1 -474.505,E2 -474.505} C_VEL
LIN {X 0,Y 608.417,Z 95.32,A -85,B 0,C 180,E1 -474.573,E2 -474.573} C_VEL
LIN {X 0,Y 608.476,Z 95.321,A -85,B 0,C 180,E1 -477.207,E2 -477.207} C_VEL
LIN {X 0,Y 608.409,Z 95.318,A -85,B 0,C 180,E1 -479.962,E2 -479.962} C_VEL
LIN {X 0,Y 608.42,Z 95.319,A -85,B 0,C 180,E1 -482.516,E2 -482.516} C_VEL
LIN {X 0,Y 608.419,Z 95.323,A -85,B 0,C 180,E1 -485.279,E2 -485.279} C_VEL
LIN {X 0,Y 608.435,Z 95.315,A -85,B 0,C 180,E1 -487.749,E2 -487.749} C_VEL
LIN {X 0,Y 608.432,Z 95.317,A -85,B 0,C 180,E1 -490.327,E2 -490.327} C_VEL
LIN {X 0,Y 608.46,Z 95.314,A -85,B 0,C 180,E1 -493.308,E2 -493.308} C_VEL
LIN {X 0,Y 608.431,Z 95.317,A -85,B 0,C 180,E1 -496.127,E2 -496.127} C_VEL
LIN {X 0,Y 608.454,Z 95.32,A -85,B 0,C 180,E1 -498.824,E2 -498.824} C_VEL
LIN {X 0,Y 608.429,Z 95.316,A -85,B 0,C 180,E1 -501.764,E2 -501.764} C_VEL
LIN {X 0,Y 608.433,Z 95.317,A -85,B 0,C 180,E1 -503.957,E2 -503.957} C_VEL
LIN {X 0,Y 608.447,Z 95.321,A -85,B 0,C 180,E1 -506.328,E2 -506.328} C_VEL
LIN {X 0,Y 608.443,Z 95.319,A -85,B 0,C 180,E1 -508.733,E2 -508.733} C_VEL
LIN {X 0,Y 608.432,Z 95.315,A -85,B 0,C 180,E1 -511.387,E2 -511.387} C_VEL
LIN {X 0,Y 608.43,Z 95.321,A -85,B 0,C 180,E1 -513.964,E2 -513.964} C_VEL
LIN {X 0,Y 608.428,Z 95.317,A -85,B 0,C 180,E1 -516.875,E2 -516.875} C_VEL
LIN {X 0,Y 608.425,Z 95.407,A -85,B 0,C 180,E1 -519.332,E2 -519.332} C_VEL
LIN {X 0,Y 608.487,Z 109.18,A -85,B 0,C 180,E1 -521.28,E2 -521.28} C_VEL
LIN {X 0,Y 608.508,Z 111.663,A -85,B 0,C 180,E1 -521.61,E2 -521.61} C_VEL
LIN {X 0,Y 608.743,Z 121.521,A -85,B 0,C 180,E1 -521.737,E2 -521.737} C_VEL
LIN {X 0,Y 608.675,Z 275.686,A -85,B 0,C 180,E1 -523.619,E2 -523.619} C_VEL
LIN {X 0,Y 608.684,Z 291.645,A -85,B 0,C 180,E1 -523.955,E2 -523.955} C_VEL
LIN {X 0,Y 608.618,Z 306.972,A -85,B 0,C 180,E1 -524.426,E2 -524.426} C_VEL
LIN {X 0,Y 608.588,Z 321.678,A -85,B 0,C 180,E1 -525.026,E2 -525.026} C_VEL
LIN {X 0,Y 608.57,Z 335.436,A -85,B 0,C 180,E1 -525.735,E2 -525.735} C_VEL
LIN {X 0,Y 608.548,Z 348.544,A -85,B 0,C 180,E1 -526.561,E2 -526.561} C_VEL
LIN {X 0,Y 608.505,Z 360.843,A -85,B 0,C 180,E1 -527.493,E2 -527.493} C_VEL
LIN {X 0,Y 608.498,Z 372.052,A -85,B 0,C 180,E1 -528.508,E2 -528.508} C_VEL
LIN {X 0,Y 608.477,Z 382.936,A -85,B 0,C 180,E1 -529.687,E2 -529.687} C_VEL
LIN {X 0,Y 608.469,Z 391.985,A -85,B 0,C 180,E1 -530.862,E2 -530.862} C_VEL
LIN {X 0,Y 608.456,Z 399.482,A -85,B 0,C 180,E1 -532.033,E2 -532.033} C_VEL
LIN {X 0,Y 608.445,Z 406.63,A -85,B 0,C 180,E1 -533.397,E2 -533.397} C_VEL
LIN {X 0,Y 608.435,Z 411.995,A -85,B 0,C 180,E1 -534.698,E2 -534.698} C_VEL
LIN {X 0,Y 608.431,Z 416.168,A -85,B 0,C 180,E1 -536.026,E2 -536.026} C_VEL
LIN {X 0,Y 608.421,Z 419.11,A -85,B 0,C 180,E1 -537.352,E2 -537.352} C_VEL
LIN {X 0,Y 608.444,Z 420.881,A -85,B 0,C 180,E1 -538.676,E2 -538.676} C_VEL
LIN {X 0,Y 608.432,Z 421.495,A -85,B 0,C 180,E1 -540,E2 -540} C_VEL
LIN {X 0,Y 608.445,Z 420.944,A -85,B 0,C 180,E1 -541.324,E2 -541.324} C_VEL
LIN {X 0,Y 608.424,Z 419.259,A -85,B 0,C 180,E1 -542.648,E2 -542.648} C_VEL
LIN {X 0,Y 608.431,Z 416.408,A -85,B 0,C 180,E1 -543.974,E2 -543.974} C_VEL
LIN {X 0,Y 608.435,Z 412.328,A -85,B 0,C 180,E1 -545.302,E2 -545.302} C_VEL
LIN {X 0,Y 608.438,Z 406.921,A -85,B 0,C 180,E1 -546.633,E2 -546.633} C_VEL
LIN {X 0,Y 608.457,Z 400.019,A -85,B 0,C 180,E1 -547.967,E2 -547.967} C_VEL
LIN {X 0,Y 608.465,Z 392.513,A -85,B 0,C 180,E1 -549.149,E2 -549.149} C_VEL
LIN {X 0,Y 607.763,Z 389.275,A -85,B 0,C 180,E1 -549.611,E2 -549.611} C_VEL
LIN {X 0,Y 602.522,Z 379.315,A -85,B 0,C 180,E1 -550.924,E2 -550.924} C_VEL
LIN {X 0,Y 601.527,Z 375.578,A -85,B 0,C 180,E1 -551.351,E2 -551.351} C_VEL
LIN {X 0,Y 601.459,Z 374.248,A -85,B 0,C 180,E1 -551.491,E2 -551.491} C_VEL
LIN {X 0,Y 601.492,Z 363.85,A -85,B 0,C 180,E1 -552.484,E2 -552.484} C_VEL
LIN {X 0,Y 601.577,Z 352.133,A -85,B 0,C 180,E1 -553.426,E2 -553.426} C_VEL
LIN {X 0,Y 601.627,Z 339.368,A -85,B 0,C 180,E1 -554.287,E2 -554.287} C_VEL
LIN {X 0,Y 601.674,Z 325.264,A -85,B 0,C 180,E1 -555.064,E2 -555.064} C_VEL
LIN {X 0,Y 601.753,Z 310.48,A -85,B 0,C 180,E1 -555.713,E2 -555.713} C_VEL
LIN {X 0,Y 601.82,Z 295.576,A -85,B 0,C 180,E1 -556.211,E2 -556.211} C_VEL
LIN {X 0,Y 601.873,Z 279.628,A -85,B 0,C 180,E1 -556.59,E2 -556.59} C_VEL
LIN {X 0,Y 601.877,Z 259.378,A -85,B 0,C 180,E1 -556.878,E2 -556.878} C_VEL
LIN {X 0,Y 601.935,Z 113.455,A -85,B 0,C 180,E1 -558.667,E2 -558.667} C_VEL
LIN {X 0,Y 601.539,Z 111.472,A -85,B 0,C 180,E1 -558.709,E2 -558.709} C_VEL
LIN {X 0,Y 601.486,Z 96.77,A -85,B 0,C 180,E1 -560.812,E2 -560.812} C_VEL
LIN {X 0,Y 601.405,Z 96.194,A -85,B 0,C 180,E1 -560.901,E2 -560.901} C_VEL
LIN {X 0,Y 601.387,Z 96.196,A -85,B 0,C 180,E1 -563.412,E2 -563.412} C_VEL
LIN {X 0,Y 601.411,Z 96.2,A -85,B 0,C 180,E1 -565.867,E2 -565.867} C_VEL
LIN {X 0,Y 601.403,Z 96.191,A -85,B 0,C 180,E1 -568.783,E2 -568.783} C_VEL
LIN {X 0,Y 601.418,Z 96.196,A -85,B 0,C 180,E1 -571.454,E2 -571.454} C_VEL
LIN {X 0,Y 601.408,Z 96.193,A -85,B 0,C 180,E1 -574.12,E2 -574.12} C_VEL
LIN {X 0,Y 601.391,Z 96.192,A -85,B 0,C 180,E1 -576.584,E2 -576.584} C_VEL
LIN {X 0,Y 601.403,Z 96.195,A -85,B 0,C 180,E1 -579.128,E2 -579.128} C_VEL
LIN {X 0,Y 601.407,Z 96.195,A -85,B 0,C 180,E1 -581.767,E2 -581.767} C_VEL
LIN {X 0,Y 601.4,Z 96.191,A -85,B 0,C 180,E1 -584.533,E2 -584.533} C_VEL
LIN {X 0,Y 601.381,Z 96.201,A -85,B 0,C 180,E1 -587.413,E2 -587.413} C_VEL
LIN {X 0,Y 601.377,Z 96.194,A -85,B 0,C 180,E1 -590.002,E2 -590.002} C_VEL
LIN {X 0,Y 601.436,Z 96.189,A -85,B 0,C 180,E1 -592.619,E2 -592.619} C_VEL
LIN {X 0,Y 601.404,Z 96.191,A -85,B 0,C 180,E1 -595.88,E2 -595.88} C_VEL
LIN {X 0,Y 601.395,Z 96.196,A -85,B 0,C 180,E1 -598.55,E2 -598.55} C_VEL
LIN {X 0,Y 601.395,Z 96.194,A -85,B 0,C 180,E1 -601.371,E2 -601.371} C_VEL
LIN {X 0,Y 601.379,Z 96.194,A -85,B 0,C 180,E1 -603.635,E2 -603.635} C_VEL
LIN {X 0,Y 601.396,Z 96.191,A -85,B 0,C 180,E1 -605.857,E2 -605.857} C_VEL
LIN {X 0,Y 601.395,Z 96.201,A -85,B 0,C 180,E1 -608.76,E2 -608.76} C_VEL
LIN {X 0,Y 601.362,Z 96.196,A -85,B 0,C 180,E1 -611.606,E2 -611.606} C_VEL
LIN {X 0,Y 601.394,Z 96.2,A -85,B 0,C 180,E1 -614.408,E2 -614.408} C_VEL
LIN {X 0,Y 601.357,Z 96.197,A -85,B 0,C 180,E1 -617.17,E2 -617.17} C_VEL
LIN {X 0,Y 601.418,Z 96.192,A -85,B 0,C 180,E1 -619.905,E2 -619.905} C_VEL
LIN {X 0,Y 601.38,Z 96.199,A -85,B 0,C 180,E1 -622.614,E2 -622.614} C_VEL
LIN {X 0,Y 601.374,Z 96.195,A -85,B 0,C 180,E1 -625.308,E2 -625.308} C_VEL
LIN {X 0,Y 601.433,Z 96.194,A -85,B 0,C 180,E1 -627.991,E2 -627.991} C_VEL
LIN {X 0,Y 601.37,Z 96.198,A -85,B 0,C 180,E1 -630.67,E2 -630.67} C_VEL
LIN {X 0,Y 601.391,Z 96.248,A -85,B 0,C 180,E1 -632.91,E2 -632.91} C_VEL
LIN {X 0,Y 601.768,Z 102.277,A -85,B 0,C 180,E1 -633.683,E2 -633.683} C_VEL
LIN {X 0,Y 601.643,Z 124.252,A -85,B 0,C 180,E1 -636.403,E2 -636.403} C_VEL
LIN {X 0,Y 601.603,Z 140.446,A -85,B 0,C 180,E1 -638.376,E2 -638.376} C_VEL
LIN {X 0,Y 602.003,Z 144.085,A -85,B 0,C 180,E1 -638.433,E2 -638.433} C_VEL
LIN {X 0,Y 601.868,Z 305.693,A -85,B 0,C 180,E1 -640.428,E2 -640.428} C_VEL
LIN {X 0,Y 601.83,Z 320.792,A -85,B 0,C 180,E1 -640.747,E2 -640.747} C_VEL
LIN {X 0,Y 601.787,Z 335.256,A -85,B 0,C 180,E1 -641.186,E2 -641.186} C_VEL
LIN {X 0,Y 601.729,Z 350.434,A -85,B 0,C 180,E1 -641.794,E2 -641.794} C_VEL
LIN {X 0,Y 601.653,Z 363.877,A -85,B 0,C 180,E1 -642.48,E2 -642.48} C_VEL
LIN {X 0,Y 601.599,Z 376.347,A -85,B 0,C 180,E1 -643.254,E2 -643.254} C_VEL
LIN {X 0,Y 601.543,Z 389.084,A -85,B 0,C 180,E1 -644.202,E2 -644.202} C_VEL
LIN {X 0,Y 601.462,Z 400.72,A -85,B 0,C 180,E1 -645.243,E2 -645.243} C_VEL
LIN {X 0,Y 601.441,Z 411.577,A -85,B 0,C 180,E1 -646.406,E2 -646.406} C_VEL
LIN {X 0,Y 601.421,Z 421.523,A -85,B 0,C 180,E1 -647.688,E2 -647.688} C_VEL
LIN {X 0,Y 601.38,Z 428.701,A -85,B 0,C 180,E1 -648.807,E2 -648.807} C_VEL
LIN {X 0,Y 601.368,Z 435.903,A -85,B 0,C 180,E1 -650.167,E2 -650.167} C_VEL
LIN {X 0,Y 601.341,Z 441.877,A -85,B 0,C 180,E1 -651.601,E2 -651.601} C_VEL
LIN {X 0,Y 601.327,Z 445.397,A -85,B 0,C 180,E1 -652.686,E2 -652.686} C_VEL
LIN {X 0,Y 601.345,Z 448.814,A -85,B 0,C 180,E1 -654.145,E2 -654.145} C_VEL
LIN {X 0,Y 601.334,Z 450.854,A -85,B 0,C 180,E1 -655.622,E2 -655.622} C_VEL
LIN {X 0,Y 601.335,Z 451.489,A -85,B 0,C 180,E1 -657.117,E2 -657.117} C_VEL
LIN {X 0,Y 601.325,Z 450.682,A -85,B 0,C 180,E1 -658.632,E2 -658.632} C_VEL
LIN {X 0,Y 601.348,Z 448.375,A -85,B 0,C 180,E1 -660.169,E2 -660.169} C_VEL
LIN {X 0,Y 601.334,Z 445.299,A -85,B 0,C 180,E1 -661.441,E2 -661.441} C_VEL
LIN {X 0,Y 601.344,Z 440.014,A -85,B 0,C 180,E1 -662.984,E2 -662.984} C_VEL
LIN {X 0,Y 601.352,Z 433.964,A -85,B 0,C 180,E1 -664.326,E2 -664.326} C_VEL
LIN {X 0,Y 601.368,Z 426.915,A -85,B 0,C 180,E1 -665.582,E2 -665.582} C_VEL
LIN {X 0,Y 601.4,Z 418.686,A -85,B 0,C 180,E1 -666.792,E2 -666.792} C_VEL
LIN {X 0,Y 601.433,Z 410.199,A -85,B 0,C 180,E1 -667.842,E2 -667.842} C_VEL
LIN {X 0,Y 601.49,Z 399.72,A -85,B 0,C 180,E1 -668.943,E2 -668.943} C_VEL
LIN {X 0,Y 601.555,Z 387.894,A -85,B 0,C 180,E1 -669.984,E2 -669.984} C_VEL
LIN {X 0,Y 601.581,Z 375.989,A -85,B 0,C 180,E1 -670.861,E2 -670.861} C_VEL
LIN {X 0,Y 601.662,Z 362.598,A -85,B 0,C 180,E1 -671.68,E2 -671.68} C_VEL
LIN {X 0,Y 601.752,Z 347.752,A -85,B 0,C 180,E1 -672.414,E2 -672.414} C_VEL
LIN {X 0,Y 601.779,Z 333.009,A -85,B 0,C 180,E1 -672.98,E2 -672.98} C_VEL
LIN {X 0,Y 601.85,Z 317.67,A -85,B 0,C 180,E1 -673.418,E2 -673.418} C_VEL
LIN {X 0,Y 601.869,Z 301.831,A -85,B 0,C 180,E1 -673.719,E2 -673.719} C_VEL
LIN {X 0,Y 601.951,Z 140.196,A -85,B 0,C 180,E1 -675.706,E2 -675.706} C_VEL
LIN {X 0,Y 601.699,Z 138.62,A -85,B 0,C 180,E1 -675.741,E2 -675.741} C_VEL
LIN {X 0,Y 601.784,Z 110.263,A -85,B 0,C 180,E1 -678.46,E2 -678.46} C_VEL
LIN {X 0,Y 601.702,Z 97.56,A -85,B 0,C 180,E1 -679.698,E2 -679.698} C_VEL
LIN {X 0,Y 601.382,Z 96.2,A -85,B 0,C 180,E1 -679.858,E2 -679.858} C_VEL
LIN {X 0,Y 601.438,Z 96.192,A -85,B 0,C 180,E1 -682.618,E2 -682.618} C_VEL
LIN {X 0,Y 601.401,Z 96.192,A -85,B 0,C 180,E1 -685.067,E2 -685.067} C_VEL
LIN {X 0,Y 601.423,Z 96.193,A -85,B 0,C 180,E1 -687.483,E2 -687.483} C_VEL
LIN {X 0,Y 601.431,Z 96.196,A -85,B 0,C 180,E1 -689.851,E2 -689.851} C_VEL
LIN {X 0,Y 601.416,Z 96.19,A -85,B 0,C 180,E1 -692.638,E2 -692.638} C_VEL
LIN {X 0,Y 601.4,Z 96.198,A -85,B 0,C 180,E1 -695.121,E2 -695.121} C_VEL
LIN {X 0,Y 601.419,Z 96.197,A -85,B 0,C 180,E1 -697.394,E2 -697.394} C_VEL
LIN {X 0,Y 601.418,Z 96.344,A -85,B 0,C 180,E1 -699.857,E2 -699.857} C_VEL
LIN {X 0,Y 601.68,Z 99.319,A -85,B 0,C 180,E1 -700.2,E2 -700.2} C_VEL
LIN {X 0,Y 601.602,Z 109.688,A -85,B 0,C 180,E1 -701.355,E2 -701.355} C_VEL
LIN {X 0,Y 601.999,Z 112.829,A -85,B 0,C 180,E1 -701.418,E2 -701.418} C_VEL
LIN {X 0,Y 601.873,Z 275.217,A -85,B 0,C 180,E1 -703.422,E2 -703.422} C_VEL
LIN {X 0,Y 601.839,Z 289.852,A -85,B 0,C 180,E1 -703.724,E2 -703.724} C_VEL
LIN {X 0,Y 601.784,Z 305.766,A -85,B 0,C 180,E1 -704.201,E2 -704.201} C_VEL
LIN {X 0,Y 601.718,Z 319.725,A -85,B 0,C 180,E1 -704.764,E2 -704.764} C_VEL
LIN {X 0,Y 601.652,Z 333.41,A -85,B 0,C 180,E1 -705.454,E2 -705.454} C_VEL
LIN {X 0,Y 601.617,Z 346.795,A -85,B 0,C 180,E1 -706.283,E2 -706.283} C_VEL
LIN {X 0,Y 601.531,Z 358.726,A -85,B 0,C 180,E1 -707.174,E2 -707.174} C_VEL
LIN {X 0,Y 601.489,Z 370.269,A -85,B 0,C 180,E1 -708.201,E2 -708.201} C_VEL
LIN {X 0,Y 601.43,Z 380,A -85,B 0,C 180,E1 -709.224,E2 -709.224} C_VEL
LIN {X 0,Y 601.428,Z 389.53,A -85,B 0,C 180,E1 -710.414,E2 -710.414} C_VEL
LIN {X 0,Y 601.377,Z 397.453,A -85,B 0,C 180,E1 -711.6,E2 -711.6} C_VEL
LIN {X 0,Y 601.368,Z 404.874,A -85,B 0,C 180,E1 -712.951,E2 -712.951} C_VEL
LIN {X 0,Y 601.373,Z 410.763,A -85,B 0,C 180,E1 -714.299,E2 -714.299} C_VEL
LIN {X 0,Y 601.328,Z 414.243,A -85,B 0,C 180,E1 -715.307,E2 -715.307} C_VEL
LIN {X 0,Y 601.336,Z 417.793,A -85,B 0,C 180,E1 -716.65,E2 -716.65} C_VEL
LIN {X 0,Y 601.343,Z 420.136,A -85,B 0,C 180,E1 -717.99,E2 -717.99} C_VEL
LIN {X 0,Y 601.334,Z 421.327,A -85,B 0,C 180,E1 -719.33,E2 -719.33} C_VEL
LIN {X 0,Y 601.335,Z 421.359,A -85,B 0,C 180,E1 -720.669,E2 -720.669} C_VEL
LIN {X 0,Y 601.343,Z 420.242,A -85,B 0,C 180,E1 -722.009,E2 -722.009} C_VEL
LIN {X 0,Y 601.339,Z 417.987,A -85,B 0,C 180,E1 -723.35,E2 -723.35} C_VEL
LIN {X 0,Y 601.328,Z 414.528,A -85,B 0,C 180,E1 -724.693,E2 -724.693} C_VEL
LIN {X 0,Y 601.358,Z 409.792,A -85,B 0,C 180,E1 -726.037,E2 -726.037} C_VEL
LIN {X 0,Y 601.365,Z 403.659,A -85,B 0,C 180,E1 -727.386,E2 -727.386} C_VEL
LIN {X 0,Y 601.389,Z 395.955,A -85,B 0,C 180,E1 -728.738,E2 -728.738} C_VEL
LIN {X 0,Y 601.428,Z 387.711,A -85,B 0,C 180,E1 -729.925,E2 -729.925} C_VEL
LIN {X 0,Y 601.445,Z 378.644,A -85,B 0,C 180,E1 -731.021,E2 -731.021} C_VEL
LIN {X 0,Y 601.514,Z 367.648,A -85,B 0,C 180,E1 -732.14,E2 -732.14} C_VEL
LIN {X 0,Y 601.57,Z 355.601,A -85,B 0,C 180,E1 -733.168,E2 -733.168} C_VEL
LIN {X 0,Y 601.632,Z 342.134,A -85,B 0,C 180,E1 -734.115,E2 -734.115} C_VEL
LIN {X 0,Y 601.656,Z 328.73,A -85,B 0,C 180,E1 -734.891,E2 -734.891} C_VEL
LIN {X 0,Y 601.741,Z 313.833,A -85,B 0,C 180,E1 -735.582,E2 -735.582} C_VEL
LIN {X 0,Y 601.817,Z 299.286,A -85,B 0,C 180,E1 -736.102,E2 -736.102} C_VEL
LIN {X 0,Y 601.853,Z 285.044,A -85,B 0,C 180,E1 -736.479,E2 -736.479} C_VEL
LIN {X 0,Y 601.885,Z 270.703,A -85,B 0,C 180,E1 -736.734,E2 -736.734} C_VEL
LIN {X 0,Y 601.937,Z 113.416,A -85,B 0,C 180,E1 -738.667,E2 -738.667} C_VEL
LIN {X 0,Y 601.538,Z 111.473,A -85,B 0,C 180,E1 -738.709,E2 -738.709} C_VEL
LIN {X 0,Y 601.485,Z 96.771,A -85,B 0,C 180,E1 -740.811,E2 -740.811} C_VEL
LIN {X 0,Y 601.408,Z 96.194,A -85,B 0,C 180,E1 -740.9,E2 -740.9} C_VEL
LIN {X 0,Y 601.387,Z 96.197,A -85,B 0,C 180,E1 -743.412,E2 -743.412} C_VEL
LIN {X 0,Y 601.411,Z 96.2,A -85,B 0,C 180,E1 -745.867,E2 -745.867} C_VEL
LIN {X 0,Y 601.402,Z 96.191,A -85,B 0,C 180,E1 -748.783,E2 -748.783} C_VEL
LIN {X 0,Y 601.416,Z 96.197,A -85,B 0,C 180,E1 -751.454,E2 -751.454} C_VEL
LIN {X 0,Y 601.406,Z 96.193,A -85,B 0,C 180,E1 -754.12,E2 -754.12} C_VEL
LIN {X 0,Y 601.389,Z 96.193,A -85,B 0,C 180,E1 -756.584,E2 -756.584} C_VEL
LIN {X 0,Y 601.4,Z 96.197,A -85,B 0,C 180,E1 -759.127,E2 -759.127} C_VEL
LIN {X 0,Y 601.4,Z 96.195,A -85,B 0,C 180,E1 -761.767,E2 -761.767} C_VEL
LIN {X 0,Y 601.397,Z 96.193,A -85,B 0,C 180,E1 -764.532,E2 -764.532} C_VEL
LIN {X 0,Y 601.373,Z 96.201,A -85,B 0,C 180,E1 -767.413,E2 -767.413} C_VEL
LIN {X 0,Y 601.374,Z 96.195,A -85,B 0,C 180,E1 -770.002,E2 -770.002} C_VEL
LIN {X 0,Y 601.432,Z 96.192,A -85,B 0,C 180,E1 -772.618,E2 -772.618} C_VEL
LIN {X 0,Y 601.396,Z 96.192,A -85,B 0,C 180,E1 -775.879,E2 -775.879} C_VEL
LIN {X 0,Y 601.39,Z 96.199,A -85,B 0,C 180,E1 -778.55,E2 -778.55} C_VEL
LIN {X 0,Y 601.383,Z 96.196,A -85,B 0,C 180,E1 -781.371,E2 -781.371} C_VEL
LIN {X 0,Y 601.381,Z 96.236,A -85,B 0,C 180,E1 -783.331,E2 -783.331} C_VEL
LIN {X 0,Y 601.933,Z 100.578,A -85,B 0,C 180,E1 -783.844,E2 -783.844} C_VEL
LIN {X 0,Y 601.863,Z 125.6,A -85,B 0,C 180,E1 -786.608,E2 -786.608} C_VEL
LIN {X 0,Y 601.74,Z 152.258,A -85,B 0,C 180,E1 -789.489,E2 -789.489} C_VEL
LIN {X 0,Y 601.653,Z 169.448,A -85,B 0,C 180,E1 -791.319,E2 -791.319} C_VEL
LIN {X 0,Y 602.035,Z 172.79,A -85,B 0,C 180,E1 -791.373,E2 -791.373} C_VEL
LIN {X 0,Y 601.885,Z 335.313,A -85,B 0,C 180,E1 -793.378,E2 -793.378} C_VEL
LIN {X 0,Y 601.86,Z 350.888,A -85,B 0,C 180,E1 -793.704,E2 -793.704} C_VEL
LIN {X 0,Y 601.797,Z 365.791,A -85,B 0,C 180,E1 -794.158,E2 -794.158} C_VEL
LIN {X 0,Y 601.723,Z 380.76,A -85,B 0,C 180,E1 -794.764,E2 -794.764} C_VEL
LIN {X 0,Y 601.658,Z 394.234,A -85,B 0,C 180,E1 -795.455,E2 -795.455} C_VEL
LIN {X 0,Y 601.617,Z 407.449,A -85,B 0,C 180,E1 -796.283,E2 -796.283} C_VEL
LIN {X 0,Y 601.531,Z 419.285,A -85,B 0,C 180,E1 -797.174,E2 -797.174} C_VEL
LIN {X 0,Y 601.488,Z 430.748,A -85,B 0,C 180,E1 -798.201,E2 -798.201} C_VEL
LIN {X 0,Y 601.43,Z 440.389,A -85,B 0,C 180,E1 -799.224,E2 -799.224} C_VEL
LIN {X 0,Y 601.428,Z 449.855,A -85,B 0,C 180,E1 -800.415,E2 -800.415} C_VEL
LIN {X 0,Y 601.369,Z 457.73,A -85,B 0,C 180,E1 -801.6,E2 -801.6} C_VEL
LIN {X 0,Y 601.367,Z 465.088,A -85,B 0,C 180,E1 -802.951,E2 -802.951} C_VEL
LIN {X 0,Y 601.373,Z 470.924,A -85,B 0,C 180,E1 -804.299,E2 -804.299} C_VEL
LIN {X 0,Y 601.33,Z 474.383,A -85,B 0,C 180,E1 -805.307,E2 -805.307} C_VEL
LIN {X 0,Y 601.337,Z 477.886,A -85,B 0,C 180,E1 -806.65,E2 -806.65} C_VEL
LIN {X 0,Y 601.343,Z 480.192,A -85,B 0,C 180,E1 -807.991,E2 -807.991} C_VEL
LIN {X 0,Y 601.335,Z 481.35,A -85,B 0,C 180,E1 -809.33,E2 -809.33} C_VEL
LIN {X 0,Y 601.335,Z 481.35,A -85,B 0,C 180,E1 -810.67,E2 -810.67} C_VEL
LIN {X 0,Y 601.343,Z 480.192,A -85,B 0,C 180,E1 -812.009,E2 -812.009} C_VEL
LIN {X 0,Y 601.337,Z 477.886,A -85,B 0,C 180,E1 -813.35,E2 -813.35} C_VEL
LIN {X 0,Y 601.33,Z 474.383,A -85,B 0,C 180,E1 -814.693,E2 -814.693} C_VEL
LIN {X 0,Y 601.357,Z 469.608,A -85,B 0,C 180,E1 -816.038,E2 -816.038} C_VEL
LIN {X 0,Y 601.365,Z 463.425,A -85,B 0,C 180,E1 -817.386,E2 -817.386} C_VEL
LIN {X 0,Y 601.388,Z 455.653,A -85,B 0,C 180,E1 -818.738,E2 -818.738} C_VEL
LIN {X 0,Y 601.427,Z 447.37,A -85,B 0,C 180,E1 -819.925,E2 -819.925} C_VEL
LIN {X 0,Y 601.46,Z 436.932,A -85,B 0,C 180,E1 -821.165,E2 -821.165} C_VEL
LIN {X 0,Y 601.514,Z 427.191,A -85,B 0,C 180,E1 -822.141,E2 -822.141} C_VEL
LIN {X 0,Y 601.57,Z 415.016,A -85,B 0,C 180,E1 -823.168,E2 -823.168} C_VEL
LIN {X 0,Y 601.606,Z 403.075,A -85,B 0,C 180,E1 -824.012,E2 -824.012} C_VEL
LIN {X 0,Y 601.65,Z 389.525,A -85,B 0,C 180,E1 -824.805,E2 -824.805} C_VEL
LIN {X 0,Y 601.771,Z 374.84,A -85,B 0,C 180,E1 -825.495,E2 -825.495} C_VEL
LIN {X 0,Y 601.803,Z 360.616,A -85,B 0,C 180,E1 -826.016,E2 -826.016} C_VEL
LIN {X 0,Y 601.845,Z 345.798,A -85,B 0,C 180,E1 -826.418,E2 -826.418} C_VEL
LIN {X 0,Y 601.855,Z 331.007,A -85,B 0,C 180,E1 -826.686,E2 -826.686} C_VEL
LIN {X 0,Y 602.005,Z 170.097,A -85,B 0,C 180,E1 -828.661,E2 -828.661} C_VEL
LIN {X 0,Y 601.7,Z 167.645,A -85,B 0,C 180,E1 -828.712,E2 -828.712} C_VEL
LIN {X 0,Y 601.811,Z 140.452,A -85,B 0,C 180,E1 -830.984,E2 -830.984} C_VEL
LIN {X 0,Y 602.004,Z 106.788,A -85,B 0,C 180,E1 -833.843,E2 -833.843} C_VEL
LIN {X 0,Y 601.958,Z 98.564,A -85,B 0,C 180,E1 -834.554,E2 -834.554} C_VEL
LIN {X 0,Y 601.382,Z 96.2,A -85,B 0,C 180,E1 -834.804,E2 -834.804} C_VEL
LIN {X 0,Y 601.407,Z 96.199,A -85,B 0,C 180,E1 -837.361,E2 -837.361} C_VEL
LIN {X 0,Y 601.371,Z 96.195,A -85,B 0,C 180,E1 -840.167,E2 -840.167} C_VEL
LIN {X 0,Y 601.393,Z 96.197,A -85,B 0,C 180,E1 -842.711,E2 -842.711} C_VEL
LIN {X 0,Y 601.379,Z 96.203,A -85,B 0,C 180,E1 -845.11,E2 -845.11} C_VEL
LIN {X 0,Y 601.43,Z 96.191,A -85,B 0,C 180,E1 -847.42,E2 -847.42} C_VEL
LIN {X 0,Y 601.374,Z 96.195,A -85,B 0,C 180,E1 -849.998,E2 -849.998} C_VEL
LIN {X 0,Y 601.38,Z 96.202,A -85,B 0,C 180,E1 -852.673,E2 -852.673} C_VEL
LIN {X 0,Y 601.398,Z 96.192,A -85,B 0,C 180,E1 -855.48,E2 -855.48} C_VEL
LIN {X 0,Y 601.411,Z 96.196,A -85,B 0,C 180,E1 -858.408,E2 -858.408} C_VEL
LIN {X 0,Y 601.399,Z 96.197,A -85,B 0,C 180,E1 -860.873,E2 -860.873} C_VEL
LIN {X 0,Y 601.388,Z 96.193,A -85,B 0,C 180,E1 -863.416,E2 -863.416} C_VEL
LIN {X 0,Y 601.411,Z 96.194,A -85,B 0,C 180,E1 -866.068,E2 -866.068} C_VEL
LIN {X 0,Y 601.393,Z 96.194,A -85,B 0,C 180,E1 -869.057,E2 -869.057} C_VEL
LIN {X 0,Y 601.392,Z 96.193,A -85,B 0,C 180,E1 -871.371,E2 -871.371} C_VEL
LIN {X 0,Y 601.41,Z 96.198,A -85,B 0,C 180,E1 -874.134,E2 -874.134} C_VEL
LIN {X 0,Y 601.383,Z 96.198,A -85,B 0,C 180,E1 -876.588,E2 -876.588} C_VEL
LIN {X 0,Y 601.4,Z 96.316,A -85,B 0,C 180,E1 -879.21,E2 -879.21} C_VEL
LIN {X 0,Y 601.549,Z 106.883,A -85,B 0,C 180,E1 -880.728,E2 -880.728} C_VEL
LIN {X 0,Y 601.506,Z 111.443,A -85,B 0,C 180,E1 -881.376,E2 -881.376} C_VEL
LIN {X 0,Y 602.013,Z 115.314,A -85,B 0,C 180,E1 -881.449,E2 -881.449} C_VEL
LIN {X 0,Y 601.863,Z 275.5,A -85,B 0,C 180,E1 -883.426,E2 -883.426} C_VEL
LIN {X 0,Y 601.841,Z 290.77,A -85,B 0,C 180,E1 -883.746,E2 -883.746} C_VEL
LIN {X 0,Y 601.784,Z 305.769,A -85,B 0,C 180,E1 -884.202,E2 -884.202} C_VEL
LIN {X 0,Y 601.717,Z 319.731,A -85,B 0,C 180,E1 -884.764,E2 -884.764} C_VEL
LIN {X 0,Y 601.652,Z 333.433,A -85,B 0,C 180,E1 -885.455,E2 -885.455} C_VEL
LIN {X 0,Y 601.617,Z 346.783,A -85,B 0,C 180,E1 -886.284,E2 -886.284} C_VEL
LIN {X 0,Y 601.541,Z 359.8,A -85,B 0,C 180,E1 -887.26,E2 -887.26} C_VEL
LIN {X 0,Y 601.489,Z 370.281,A -85,B 0,C 180,E1 -888.201,E2 -888.201} C_VEL
LIN {X 0,Y 601.43,Z 380.005,A -85,B 0,C 180,E1 -889.224,E2 -889.224} C_VEL
LIN {X 0,Y 601.428,Z 389.525,A -85,B 0,C 180,E1 -890.415,E2 -890.415} C_VEL
LIN {X 0,Y 601.4,Z 398.478,A -85,B 0,C 180,E1 -891.77,E2 -891.77} C_VEL
LIN {X 0,Y 601.368,Z 404.875,A -85,B 0,C 180,E1 -892.952,E2 -892.952} C_VEL
LIN {X 0,Y 601.373,Z 410.762,A -85,B 0,C 180,E1 -894.299,E2 -894.299} C_VEL
LIN {X 0,Y 601.328,Z 414.247,A -85,B 0,C 180,E1 -895.307,E2 -895.307} C_VEL
LIN {X 0,Y 601.336,Z 417.788,A -85,B 0,C 180,E1 -896.65,E2 -896.65} C_VEL
LIN {X 0,Y 601.343,Z 420.143,A -85,B 0,C 180,E1 -897.991,E2 -897.991} C_VEL
LIN {X 0,Y 601.334,Z 421.332,A -85,B 0,C 180,E1 -899.331,E2 -899.331} C_VEL
LIN {X 0,Y 601.335,Z 421.36,A -85,B 0,C 180,E1 -900.67,E2 -900.67} C_VEL
LIN {X 0,Y 601.343,Z 420.248,A -85,B 0,C 180,E1 -902.01,E2 -902.01} C_VEL
LIN {X 0,Y 601.339,Z 417.981,A -85,B 0,C 180,E1 -903.35,E2 -903.35} C_VEL
LIN {X 0,Y 601.33,Z 414.529,A -85,B 0,C 180,E1 -904.693,E2 -904.693} C_VEL
LIN {X 0,Y 601.358,Z 409.792,A -85,B 0,C 180,E1 -906.038,E2 -906.038} C_VEL
LIN {X 0,Y 601.366,Z 403.664,A -85,B 0,C 180,E1 -907.386,E2 -907.386} C_VEL
LIN {X 0,Y 601.389,Z 395.941,A -85,B 0,C 180,E1 -908.739,E2 -908.739} C_VEL
LIN {X 0,Y 601.428,Z 387.695,A -85,B 0,C 180,E1 -909.925,E2 -909.925} C_VEL
LIN {X 0,Y 601.443,Z 377.352,A -85,B 0,C 180,E1 -911.164,E2 -911.164} C_VEL
LIN {X 0,Y 601.459,Z 374.248,A -85,B 0,C 180,E1 -911.491,E2 -911.491} C_VEL
LIN {X 0,Y 600.84,Z 370.294,A -85,B 0,C 180,E1 -911.906,E2 -911.906} C_VEL
LIN {X 0,Y 598.052,Z 363.784,A -85,B 0,C 180,E1 -912.57,E2 -912.57} C_VEL
LIN {X 0,Y 595.245,Z 356.933,A -85,B 0,C 180,E1 -913.203,E2 -913.203} C_VEL
LIN {X 0,Y 594.595,Z 352.406,A -85,B 0,C 180,E1 -913.566,E2 -913.566} C_VEL
LIN {X 0,Y 594.696,Z 339.367,A -85,B 0,C 180,E1 -914.457,E2 -914.457} C_VEL
LIN {X 0,Y 594.786,Z 326.987,A -85,B 0,C 180,E1 -915.155,E2 -915.155} C_VEL
LIN {X 0,Y 594.91,Z 312.72,A -85,B 0,C 180,E1 -915.81,E2 -915.81} C_VEL
LIN {X 0,Y 594.992,Z 297.784,A -85,B 0,C 180,E1 -916.336,E2 -916.336} C_VEL
LIN {X 0,Y 595.055,Z 282.792,A -85,B 0,C 180,E1 -916.724,E2 -916.724} C_VEL
LIN {X 0,Y 595.1,Z 265.611,A -85,B 0,C 180,E1 -916.998,E2 -916.998} C_VEL
LIN {X 0,Y 595.219,Z 114.692,A -85,B 0,C 180,E1 -918.869,E2 -918.869} C_VEL
LIN {X 0,Y 594.577,Z 111.5,A -85,B 0,C 180,E1 -918.932,E2 -918.932} C_VEL
LIN {X 0,Y 594.622,Z 98.794,A -85,B 0,C 180,E1 -920.768,E2 -920.768} C_VEL
LIN {X 0,Y 594.373,Z 97.072,A -85,B 0,C 180,E1 -921.042,E2 -921.042} C_VEL
LIN {X 0,Y 594.359,Z 97.077,A -85,B 0,C 180,E1 -923.706,E2 -923.706} C_VEL
LIN {X 0,Y 594.361,Z 97.075,A -85,B 0,C 180,E1 -926.018,E2 -926.018} C_VEL
LIN {X 0,Y 594.354,Z 97.072,A -85,B 0,C 180,E1 -928.229,E2 -928.229} C_VEL
LIN {X 0,Y 594.365,Z 97.068,A -85,B 0,C 180,E1 -930.561,E2 -930.561} C_VEL
LIN {X 0,Y 594.373,Z 97.068,A -85,B 0,C 180,E1 -932.951,E2 -932.951} C_VEL
LIN {X 0,Y 594.327,Z 97.08,A -85,B 0,C 180,E1 -935.411,E2 -935.411} C_VEL
LIN {X 0,Y 594.369,Z 97.07,A -85,B 0,C 180,E1 -937.942,E2 -937.942} C_VEL
LIN {X 0,Y 594.375,Z 97.068,A -85,B 0,C 180,E1 -940.822,E2 -940.822} C_VEL
LIN {X 0,Y 594.346,Z 97.072,A -85,B 0,C 180,E1 -943.837,E2 -943.837} C_VEL
LIN {X 0,Y 594.346,Z 97.07,A -85,B 0,C 180,E1 -946.699,E2 -946.699} C_VEL
LIN {X 0,Y 594.36,Z 97.074,A -85,B 0,C 180,E1 -949.432,E2 -949.432} C_VEL
LIN {X 0,Y 594.383,Z 97.066,A -85,B 0,C 180,E1 -952.393,E2 -952.393} C_VEL
LIN {X 0,Y 594.368,Z 97.071,A -85,B 0,C 180,E1 -955.419,E2 -955.419} C_VEL
LIN {X 0,Y 594.344,Z 97.07,A -85,B 0,C 180,E1 -957.851,E2 -957.851} C_VEL
LIN {X 0,Y 594.337,Z 97.071,A -85,B 0,C 180,E1 -960.222,E2 -960.222} C_VEL
LIN {X 0,Y 594.365,Z 97.071,A -85,B 0,C 180,E1 -963.299,E2 -963.299} C_VEL
LIN {X 0,Y 594.335,Z 97.071,A -85,B 0,C 180,E1 -965.579,E2 -965.579} C_VEL
LIN {X 0,Y 594.352,Z 97.076,A -85,B 0,C 180,E1 -968.496,E2 -968.496} C_VEL
LIN {X 0,Y 594.344,Z 97.071,A -85,B 0,C 180,E1 -971.381,E2 -971.381} C_VEL
LIN {X 0,Y 594.339,Z 97.075,A -85,B 0,C 180,E1 -974.218,E2 -974.218} C_VEL
LIN {X 0,Y 594.313,Z 97.076,A -85,B 0,C 180,E1 -977.016,E2 -977.016} C_VEL
LIN {X 0,Y 594.367,Z 97.068,A -85,B 0,C 180,E1 -979.094,E2 -979.094} C_VEL
LIN {X 0,Y 594.371,Z 97.069,A -85,B 0,C 180,E1 -981.843,E2 -981.843} C_VEL
LIN {X 0,Y 594.366,Z 97.073,A -85,B 0,C 180,E1 -984.572,E2 -984.572} C_VEL
LIN {X 0,Y 594.364,Z 97.069,A -85,B 0,C 180,E1 -987.289,E2 -987.289} C_VEL
LIN {X 0,Y 594.413,Z 97.071,A -85,B 0,C 180,E1 -990,E2 -990} C_VEL
LIN {X 0,Y 594.349,Z 97.076,A -85,B 0,C 180,E1 -992.711,E2 -992.711} C_VEL
LIN {X 0,Y 594.897,Z 100.861,A -85,B 0,C 180,E1 -993.217,E2 -993.217} C_VEL
LIN {X 0,Y 594.725,Z 123.877,A -85,B 0,C 180,E1 -996.105,E2 -996.105} C_VEL
LIN {X 0,Y 594.7,Z 140.606,A -85,B 0,C 180,E1 -998.153,E2 -998.153} C_VEL
LIN {X 0,Y 595.268,Z 143.613,A -85,B 0,C 180,E1 -998.209,E2 -998.209} C_VEL
LIN {X 0,Y 595.071,Z 306.536,A -85,B 0,C 180,E1 -1000.247,E2 -1000.247} C_VEL
LIN {X 0,Y 595.004,Z 321.352,A -85,B 0,C 180,E1 -1000.571,E2 -1000.571} C_VEL
LIN {X 0,Y 594.935,Z 335.248,A -85,B 0,C 180,E1 -1000.998,E2 -1000.998} C_VEL
LIN {X 0,Y 594.865,Z 349.835,A -85,B 0,C 180,E1 -1001.586,E2 -1001.586} C_VEL
LIN {X 0,Y 594.731,Z 363.419,A -85,B 0,C 180,E1 -1002.281,E2 -1002.281} C_VEL
LIN {X 0,Y 594.659,Z 375.965,A -85,B 0,C 180,E1 -1003.063,E2 -1003.063} C_VEL
LIN {X 0,Y 594.564,Z 388.596,A -85,B 0,C 180,E1 -1004.009,E2 -1004.009} C_VEL
LIN {X 0,Y 594.467,Z 400.451,A -85,B 0,C 180,E1 -1005.076,E2 -1005.076} C_VEL
LIN {X 0,Y 594.422,Z 410.305,A -85,B 0,C 180,E1 -1006.132,E2 -1006.132} C_VEL
LIN {X 0,Y 594.352,Z 420.064,A -85,B 0,C 180,E1 -1007.372,E2 -1007.372} C_VEL
LIN {X 0,Y 594.304,Z 428.181,A -85,B 0,C 180,E1 -1008.62,E2 -1008.62} C_VEL
LIN {X 0,Y 594.287,Z 434.05,A -85,B 0,C 180,E1 -1009.697,E2 -1009.697} C_VEL
LIN {X 0,Y 594.272,Z 439.414,A -85,B 0,C 180,E1 -1010.888,E2 -1010.888} C_VEL
LIN {X 0,Y 594.269,Z 444.199,A -85,B 0,C 180,E1 -1012.237,E2 -1012.237} C_VEL
LIN {X 0,Y 594.223,Z 448.013,A -85,B 0,C 180,E1 -1013.711,E2 -1013.711} C_VEL
LIN {X 0,Y 594.218,Z 450.407,A -85,B 0,C 180,E1 -1015.2,E2 -1015.2} C_VEL
LIN {X 0,Y 594.226,Z 451.429,A -85,B 0,C 180,E1 -1016.707,E2 -1016.707} C_VEL
LIN {X 0,Y 594.254,Z 451.401,A -85,B 0,C 180,E1 -1017.501,E2 -1017.501} C_VEL
LIN {X 0,Y 594.25,Z 450.274,A -85,B 0,C 180,E1 -1019.006,E2 -1019.006} C_VEL
LIN {X 0,Y 594.232,Z 447.613,A -85,B 0,C 180,E1 -1020.568,E2 -1020.568} C_VEL
LIN {X 0,Y 594.24,Z 444.924,A -85,B 0,C 180,E1 -1021.62,E2 -1021.62} C_VEL
LIN {X 0,Y 594.261,Z 440.398,A -85,B 0,C 180,E1 -1022.958,E2 -1022.958} C_VEL
LIN {X 0,Y 594.276,Z 434.363,A -85,B 0,C 180,E1 -1024.329,E2 -1024.329} C_VEL
LIN {X 0,Y 594.312,Z 427.296,A -85,B 0,C 180,E1 -1025.62,E2 -1025.62} C_VEL
LIN {X 0,Y 594.354,Z 418.6,A -85,B 0,C 180,E1 -1026.921,E2 -1026.921} C_VEL
LIN {X 0,Y 594.412,Z 410.474,A -85,B 0,C 180,E1 -1027.939,E2 -1027.939} C_VEL
LIN {X 0,Y 594.479,Z 400.44,A -85,B 0,C 180,E1 -1029.015,E2 -1029.015} C_VEL
LIN {X 0,Y 594.586,Z 387.96,A -85,B 0,C 180,E1 -1030.133,E2 -1030.133} C_VEL
LIN {X 0,Y 594.626,Z 376.105,A -85,B 0,C 180,E1 -1031.018,E2 -1031.018} C_VEL
LIN {X 0,Y 594.742,Z 363.886,A -85,B 0,C 180,E1 -1031.782,E2 -1031.782} C_VEL
LIN {X 0,Y 594.842,Z 350.243,A -85,B 0,C 180,E1 -1032.486,E2 -1032.486} C_VEL
LIN {X 0,Y 594.938,Z 335.918,A -85,B 0,C 180,E1 -1033.069,E2 -1033.069} C_VEL
LIN {X 0,Y 595.022,Z 320.717,A -85,B 0,C 180,E1 -1033.535,E2 -1033.535} C_VEL
LIN {X 0,Y 595.098,Z 305.978,A -85,B 0,C 180,E1 -1033.852,E2 -1033.852} C_VEL
LIN {X 0,Y 595.215,Z 140.994,A -85,B 0,C 180,E1 -1035.915,E2 -1035.915} C_VEL
LIN {X 0,Y 594.829,Z 138.489,A -85,B 0,C 180,E1 -1035.978,E2 -1035.978} C_VEL
LIN {X 0,Y 595.001,Z 108.428,A -85,B 0,C 180,E1 -1038.896,E2 -1038.896} C_VEL
LIN {X 0,Y 595.034,Z 100.237,A -85,B 0,C 180,E1 -1039.701,E2 -1039.701} C_VEL
LIN {X 0,Y 594.365,Z 97.076,A -85,B 0,C 180,E1 -1040.046,E2 -1040.046} C_VEL
LIN {X 0,Y 594.383,Z 97.068,A -85,B 0,C 180,E1 -1042.913,E2 -1042.913} C_VEL
LIN {X 0,Y 594.379,Z 97.074,A -85,B 0,C 180,E1 -1045.862,E2 -1045.862} C_VEL
LIN {X 0,Y 594.372,Z 97.068,A -85,B 0,C 180,E1 -1048.65,E2 -1048.65} C_VEL
LIN {X 0,Y 594.386,Z 97.067,A -85,B 0,C 180,E1 -1051.042,E2 -1051.042} C_VEL
LIN {X 0,Y 594.384,Z 97.069,A -85,B 0,C 180,E1 -1053.978,E2 -1053.978} C_VEL
LIN {X 0,Y 594.385,Z 97.067,A -85,B 0,C 180,E1 -1056.295,E2 -1056.295} C_VEL
LIN {X 0,Y 594.397,Z 97.073,A -85,B 0,C 180,E1 -1059.224,E2 -1059.224} C_VEL
LIN {X 0,Y 594.396,Z 97.143,A -85,B 0,C 180,E1 -1059.699,E2 -1059.699} C_VEL
LIN {X 0,Y 594.79,Z 100.911,A -85,B 0,C 180,E1 -1060.141,E2 -1060.141} C_VEL
LIN {X 0,Y 594.71,Z 109.781,A -85,B 0,C 180,E1 -1061.141,E2 -1061.141} C_VEL
LIN {X 0,Y 595.287,Z 113.87,A -85,B 0,C 180,E1 -1061.213,E2 -1061.213} C_VEL
LIN {X 0,Y 595.067,Z 275.184,A -85,B 0,C 180,E1 -1063.227,E2 -1063.227} C_VEL
LIN {X 0,Y 595.023,Z 289.875,A -85,B 0,C 180,E1 -1063.532,E2 -1063.532} C_VEL
LIN {X 0,Y 594.947,Z 305.772,A -85,B 0,C 180,E1 -1064.015,E2 -1064.015} C_VEL
LIN {X 0,Y 594.839,Z 319.715,A -85,B 0,C 180,E1 -1064.583,E2 -1064.583} C_VEL
LIN {X 0,Y 594.727,Z 333.421,A -85,B 0,C 180,E1 -1065.281,E2 -1065.281} C_VEL
LIN {X 0,Y 594.682,Z 346.149,A -85,B 0,C 180,E1 -1066.075,E2 -1066.075} C_VEL
LIN {X 0,Y 594.56,Z 358.734,A -85,B 0,C 180,E1 -1067.021,E2 -1067.021} C_VEL
LIN {X 0,Y 594.466,Z 370.27,A -85,B 0,C 180,E1 -1068.06,E2 -1068.06} C_VEL
LIN {X 0,Y 594.401,Z 381.498,A -85,B 0,C 180,E1 -1069.267,E2 -1069.267} C_VEL
LIN {X 0,Y 594.342,Z 390.776,A -85,B 0,C 180,E1 -1070.471,E2 -1070.471} C_VEL
LIN {X 0,Y 594.321,Z 398.463,A -85,B 0,C 180,E1 -1071.671,E2 -1071.671} C_VEL
LIN {X 0,Y 594.293,Z 404.879,A -85,B 0,C 180,E1 -1072.867,E2 -1072.867} C_VEL
LIN {X 0,Y 594.299,Z 410.769,A -85,B 0,C 180,E1 -1074.231,E2 -1074.231} C_VEL
LIN {X 0,Y 594.231,Z 414.247,A -85,B 0,C 180,E1 -1075.251,E2 -1075.251} C_VEL
LIN {X 0,Y 594.256,Z 417.798,A -85,B 0,C 180,E1 -1076.61,E2 -1076.61} C_VEL
LIN {X 0,Y 594.241,Z 420.135,A -85,B 0,C 180,E1 -1077.966,E2 -1077.966} C_VEL
LIN {X 0,Y 594.235,Z 421.319,A -85,B 0,C 180,E1 -1079.322,E2 -1079.322} C_VEL
LIN {X 0,Y 594.236,Z 421.351,A -85,B 0,C 180,E1 -1080.677,E2 -1080.677} C_VEL
LIN {X 0,Y 594.242,Z 420.24,A -85,B 0,C 180,E1 -1082.033,E2 -1082.033} C_VEL
LIN {X 0,Y 594.258,Z 417.989,A -85,B 0,C 180,E1 -1083.39,E2 -1083.39} C_VEL
LIN {X 0,Y 594.231,Z 414.528,A -85,B 0,C 180,E1 -1084.749,E2 -1084.749} C_VEL
LIN {X 0,Y 594.279,Z 409.783,A -85,B 0,C 180,E1 -1086.11,E2 -1086.11} C_VEL
LIN {X 0,Y 594.287,Z 403.646,A -85,B 0,C 180,E1 -1087.474,E2 -1087.474} C_VEL
LIN {X 0,Y 594.332,Z 395.952,A -85,B 0,C 180,E1 -1088.843,E2 -1088.843} C_VEL
LIN {X 0,Y 594.387,Z 387.706,A -85,B 0,C 180,E1 -1090.044,E2 -1090.044} C_VEL
LIN {X 0,Y 594.431,Z 377.952,A -85,B 0,C 180,E1 -1091.229,E2 -1091.229} C_VEL
LIN {X 0,Y 594.514,Z 367.632,A -85,B 0,C 180,E1 -1092.285,E2 -1092.285} C_VEL
LIN {X 0,Y 594.579,Z 355.595,A -85,B 0,C 180,E1 -1093.326,E2 -1093.326} C_VEL
LIN {X 0,Y 594.687,Z 342.064,A -85,B 0,C 180,E1 -1094.286,E2 -1094.286} C_VEL
LIN {X 0,Y 594.772,Z 328.7,A -85,B 0,C 180,E1 -1095.067,E2 -1095.067} C_VEL
LIN {X 0,Y 594.891,Z 313.818,A -85,B 0,C 180,E1 -1095.766,E2 -1095.766} C_VEL
LIN {X 0,Y 594.984,Z 299.232,A -85,B 0,C 180,E1 -1096.292,E2 -1096.292} C_VEL
LIN {X 0,Y 595.037,Z 285.626,A -85,B 0,C 180,E1 -1096.658,E2 -1096.658} C_VEL
LIN {X 0,Y 595.073,Z 271.496,A -85,B 0,C 180,E1 -1096.919,E2 -1096.919} C_VEL
LIN {X 0,Y 595.225,Z 114.724,A -85,B 0,C 180,E1 -1098.869,E2 -1098.869} C_VEL
LIN {X 0,Y 594.579,Z 111.502,A -85,B 0,C 180,E1 -1098.932,E2 -1098.932} C_VEL
LIN {X 0,Y 594.621,Z 98.798,A -85,B 0,C 180,E1 -1100.767,E2 -1100.767} C_VEL
LIN {X 0,Y 594.372,Z 97.072,A -85,B 0,C 180,E1 -1101.042,E2 -1101.042} C_VEL
LIN {X 0,Y 594.358,Z 97.078,A -85,B 0,C 180,E1 -1103.705,E2 -1103.705} C_VEL
LIN {X 0,Y 594.361,Z 97.075,A -85,B 0,C 180,E1 -1106.017,E2 -1106.017} C_VEL
LIN {X 0,Y 594.353,Z 97.073,A -85,B 0,C 180,E1 -1108.228,E2 -1108.228} C_VEL
LIN {X 0,Y 594.362,Z 97.069,A -85,B 0,C 180,E1 -1110.561,E2 -1110.561} C_VEL
LIN {X 0,Y 594.371,Z 97.069,A -85,B 0,C 180,E1 -1112.95,E2 -1112.95} C_VEL
LIN {X 0,Y 594.325,Z 97.082,A -85,B 0,C 180,E1 -1115.411,E2 -1115.411} C_VEL
LIN {X 0,Y 594.365,Z 97.071,A -85,B 0,C 180,E1 -1117.942,E2 -1117.942} C_VEL
LIN {X 0,Y 594.372,Z 97.069,A -85,B 0,C 180,E1 -1120.821,E2 -1120.821} C_VEL
LIN {X 0,Y 594.343,Z 97.073,A -85,B 0,C 180,E1 -1123.837,E2 -1123.837} C_VEL
LIN {X 0,Y 594.342,Z 97.074,A -85,B 0,C 180,E1 -1126.698,E2 -1126.698} C_VEL
LIN {X 0,Y 594.357,Z 97.074,A -85,B 0,C 180,E1 -1129.432,E2 -1129.432} C_VEL
LIN {X 0,Y 594.379,Z 97.068,A -85,B 0,C 180,E1 -1132.393,E2 -1132.393} C_VEL
LIN {X 0,Y 594.358,Z 97.072,A -85,B 0,C 180,E1 -1135.418,E2 -1135.418} C_VEL
LIN {X 0,Y 594.335,Z 97.072,A -85,B 0,C 180,E1 -1137.851,E2 -1137.851} C_VEL
LIN {X 0,Y 594.331,Z 97.076,A -85,B 0,C 180,E1 -1140.221,E2 -1140.221} C_VEL
LIN {X 0,Y 594.384,Z 97.202,A -85,B 0,C 180,E1 -1143.134,E2 -1143.134} C_VEL
LIN {X 0,Y 595.152,Z 101.913,A -85,B 0,C 180,E1 -1143.679,E2 -1143.679} C_VEL
LIN {X 0,Y 595.048,Z 125.6,A -85,B 0,C 180,E1 -1146.324,E2 -1146.324} C_VEL
LIN {X 0,Y 594.871,Z 150.864,A -85,B 0,C 180,E1 -1149.09,E2 -1149.09} C_VEL
LIN {X 0,Y 594.739,Z 169.456,A -85,B 0,C 180,E1 -1151.094,E2 -1151.094} C_VEL
LIN {X 0,Y 595.329,Z 173.058,A -85,B 0,C 180,E1 -1151.159,E2 -1151.159} C_VEL
LIN {X 0,Y 595.08,Z 336.411,A -85,B 0,C 180,E1 -1153.2,E2 -1153.2} C_VEL
LIN {X 0,Y 595.017,Z 351.707,A -85,B 0,C 180,E1 -1153.532,E2 -1153.532} C_VEL
LIN {X 0,Y 594.944,Z 367.044,A -85,B 0,C 180,E1 -1154.015,E2 -1154.015} C_VEL
LIN {X 0,Y 594.863,Z 380.763,A -85,B 0,C 180,E1 -1154.584,E2 -1154.584} C_VEL
LIN {X 0,Y 594.732,Z 394.237,A -85,B 0,C 180,E1 -1155.282,E2 -1155.282} C_VEL
LIN {X 0,Y 594.681,Z 406.793,A -85,B 0,C 180,E1 -1156.075,E2 -1156.075} C_VEL
LIN {X 0,Y 594.56,Z 419.286,A -85,B 0,C 180,E1 -1157.021,E2 -1157.021} C_VEL
LIN {X 0,Y 594.465,Z 430.748,A -85,B 0,C 180,E1 -1158.06,E2 -1158.06} C_VEL
LIN {X 0,Y 594.388,Z 440.389,A -85,B 0,C 180,E1 -1159.095,E2 -1159.095} C_VEL
LIN {X 0,Y 594.366,Z 449.856,A -85,B 0,C 180,E1 -1160.3,E2 -1160.3} C_VEL
LIN {X 0,Y 594.312,Z 457.731,A -85,B 0,C 180,E1 -1161.499,E2 -1161.499} C_VEL
LIN {X 0,Y 594.291,Z 465.088,A -85,B 0,C 180,E1 -1162.867,E2 -1162.867} C_VEL
LIN {X 0,Y 594.299,Z 470.924,A -85,B 0,C 180,E1 -1164.231,E2 -1164.231} C_VEL
LIN {X 0,Y 594.232,Z 474.384,A -85,B 0,C 180,E1 -1165.251,E2 -1165.251} C_VEL
LIN {X 0,Y 594.257,Z 477.887,A -85,B 0,C 180,E1 -1166.61,E2 -1166.61} C_VEL
LIN {X 0,Y 594.241,Z 480.193,A -85,B 0,C 180,E1 -1167.967,E2 -1167.967} C_VEL
LIN {X 0,Y 594.235,Z 481.35,A -85,B 0,C 180,E1 -1169.322,E2 -1169.322} C_VEL
LIN {X 0,Y 594.235,Z 481.35,A -85,B 0,C 180,E1 -1170.678,E2 -1170.678} C_VEL
LIN {X 0,Y 594.241,Z 480.192,A -85,B 0,C 180,E1 -1172.033,E2 -1172.033} C_VEL
LIN {X 0,Y 594.257,Z 477.886,A -85,B 0,C 180,E1 -1173.39,E2 -1173.39} C_VEL
LIN {X 0,Y 594.232,Z 474.384,A -85,B 0,C 180,E1 -1174.749,E2 -1174.749} C_VEL
LIN {X 0,Y 594.279,Z 469.608,A -85,B 0,C 180,E1 -1176.11,E2 -1176.11} C_VEL
LIN {X 0,Y 594.287,Z 463.424,A -85,B 0,C 180,E1 -1177.475,E2 -1177.475} C_VEL
LIN {X 0,Y 594.331,Z 455.651,A -85,B 0,C 180,E1 -1178.843,E2 -1178.843} C_VEL
LIN {X 0,Y 594.387,Z 447.37,A -85,B 0,C 180,E1 -1180.044,E2 -1180.044} C_VEL
LIN {X 0,Y 594.433,Z 437.559,A -85,B 0,C 180,E1 -1181.231,E2 -1181.231} C_VEL
LIN {X 0,Y 594.53,Z 427.191,A -85,B 0,C 180,E1 -1182.285,E2 -1182.285} C_VEL
LIN {X 0,Y 594.581,Z 415.017,A -85,B 0,C 180,E1 -1183.326,E2 -1183.326} C_VEL
LIN {X 0,Y 594.694,Z 403.072,A -85,B 0,C 180,E1 -1184.178,E2 -1184.178} C_VEL
LIN {X 0,Y 594.751,Z 389.521,A -85,B 0,C 180,E1 -1184.981,E2 -1184.981} C_VEL
LIN {X 0,Y 594.913,Z 374.837,A -85,B 0,C 180,E1 -1185.678,E2 -1185.678} C_VEL
LIN {X 0,Y 594.986,Z 360.615,A -85,B 0,C 180,E1 -1186.204,E2 -1186.204} C_VEL
LIN {X 0,Y 595.043,Z 346.226,A -85,B 0,C 180,E1 -1186.6,E2 -1186.6} C_VEL
LIN {X 0,Y 595.055,Z 331.007,A -85,B 0,C 180,E1 -1186.882,E2 -1186.882} C_VEL
LIN {X 0,Y 595.281,Z 170.622,A -85,B 0,C 180,E1 -1188.873,E2 -1188.873} C_VEL
LIN {X 0,Y 594.838,Z 167.557,A -85,B 0,C 180,E1 -1188.943,E2 -1188.943} C_VEL
LIN {X 0,Y 594.988,Z 140.872,A -85,B 0,C 180,E1 -1191.2,E2 -1191.2} C_VEL
LIN {X 0,Y 595.262,Z 109.976,A -85,B 0,C 180,E1 -1193.852,E2 -1193.852} C_VEL
LIN {X 0,Y 595.132,Z 100.15,A -85,B 0,C 180,E1 -1194.716,E2 -1194.716} C_VEL
LIN {X 0,Y 594.351,Z 97.078,A -85,B 0,C 180,E1 -1195.039,E2 -1195.039} C_VEL
LIN {X 0,Y 594.342,Z 97.077,A -85,B 0,C 180,E1 -1197.518,E2 -1197.518} C_VEL
LIN {X 0,Y 594.334,Z 97.074,A -85,B 0,C 180,E1 -1199.779,E2 -1199.779} C_VEL
LIN {X 0,Y 594.339,Z 97.071,A -85,B 0,C 180,E1 -1202.149,E2 -1202.149} C_VEL
LIN {X 0,Y 594.363,Z 97.071,A -85,B 0,C 180,E1 -1204.581,E2 -1204.581} C_VEL
LIN {X 0,Y 594.38,Z 97.067,A -85,B 0,C 180,E1 -1207.607,E2 -1207.607} C_VEL
LIN {X 0,Y 594.358,Z 97.074,A -85,B 0,C 180,E1 -1210.568,E2 -1210.568} C_VEL
LIN {X 0,Y 594.343,Z 97.073,A -85,B 0,C 180,E1 -1213.302,E2 -1213.302} C_VEL
LIN {X 0,Y 594.343,Z 97.072,A -85,B 0,C 180,E1 -1216.163,E2 -1216.163} C_VEL
LIN {X 0,Y 594.372,Z 97.069,A -85,B 0,C 180,E1 -1219.179,E2 -1219.179} C_VEL
LIN {X 0,Y 594.364,Z 97.071,A -85,B 0,C 180,E1 -1222.058,E2 -1222.058} C_VEL
LIN {X 0,Y 594.324,Z 97.08,A -85,B 0,C 180,E1 -1224.68,E2 -1224.68} C_VEL
LIN {X 0,Y 594.369,Z 97.069,A -85,B 0,C 180,E1 -1227.09,E2 -1227.09} C_VEL
LIN {X 0,Y 594.364,Z 97.069,A -85,B 0,C 180,E1 -1229.676,E2 -1229.676} C_VEL
LIN {X 0,Y 594.376,Z 97.073,A -85,B 0,C 180,E1 -1232.539,E2 -1232.539} C_VEL
LIN {X 0,Y 594.368,Z 97.07,A -85,B 0,C 180,E1 -1234.807,E2 -1234.807} C_VEL
LIN {X 0,Y 594.344,Z 97.075,A -85,B 0,C 180,E1 -1237.766,E2 -1237.766} C_VEL
LIN {X 0,Y 594.388,Z 97.204,A -85,B 0,C 180,E1 -1239.082,E2 -1239.082} C_VEL
LIN {X 0,Y 594.631,Z 105.643,A -85,B 0,C 180,E1 -1240.315,E2 -1240.315} C_VEL
LIN {X 0,Y 594.574,Z 111.466,A -85,B 0,C 180,E1 -1241.153,E2 -1241.153} C_VEL
LIN {X 0,Y 595.292,Z 115.79,A -85,B 0,C 180,E1 -1241.237,E2 -1241.237} C_VEL
LIN {X 0,Y 595.062,Z 275.483,A -85,B 0,C 180,E1 -1243.231,E2 -1243.231} C_VEL
LIN {X 0,Y 595.029,Z 290.786,A -85,B 0,C 180,E1 -1243.555,E2 -1243.555} C_VEL
LIN {X 0,Y 594.954,Z 305.761,A -85,B 0,C 180,E1 -1244.015,E2 -1244.015} C_VEL
LIN {X 0,Y 594.839,Z 319.741,A -85,B 0,C 180,E1 -1244.584,E2 -1244.584} C_VEL
LIN {X 0,Y 594.734,Z 333.452,A -85,B 0,C 180,E1 -1245.282,E2 -1245.282} C_VEL
LIN {X 0,Y 594.682,Z 346.13,A -85,B 0,C 180,E1 -1246.075,E2 -1246.075} C_VEL
LIN {X 0,Y 594.56,Z 358.754,A -85,B 0,C 180,E1 -1247.021,E2 -1247.021} C_VEL
LIN {X 0,Y 594.466,Z 370.285,A -85,B 0,C 180,E1 -1248.06,E2 -1248.06} C_VEL
LIN {X 0,Y 594.401,Z 381.504,A -85,B 0,C 180,E1 -1249.268,E2 -1249.268} C_VEL
LIN {X 0,Y 594.341,Z 390.766,A -85,B 0,C 180,E1 -1250.471,E2 -1250.471} C_VEL
LIN {X 0,Y 594.321,Z 398.485,A -85,B 0,C 180,E1 -1251.671,E2 -1251.671} C_VEL
LIN {X 0,Y 594.292,Z 404.879,A -85,B 0,C 180,E1 -1252.867,E2 -1252.867} C_VEL
LIN {X 0,Y 594.299,Z 410.766,A -85,B 0,C 180,E1 -1254.231,E2 -1254.231} C_VEL
LIN {X 0,Y 594.231,Z 414.253,A -85,B 0,C 180,E1 -1255.251,E2 -1255.251} C_VEL
LIN {X 0,Y 594.256,Z 417.789,A -85,B 0,C 180,E1 -1256.61,E2 -1256.61} C_VEL
LIN {X 0,Y 594.241,Z 420.147,A -85,B 0,C 180,E1 -1257.967,E2 -1257.967} C_VEL
LIN {X 0,Y 594.235,Z 421.327,A -85,B 0,C 180,E1 -1259.323,E2 -1259.323} C_VEL
LIN {X 0,Y 594.236,Z 421.355,A -85,B 0,C 180,E1 -1260.678,E2 -1260.678} C_VEL
LIN {X 0,Y 594.242,Z 420.251,A -85,B 0,C 180,E1 -1262.034,E2 -1262.034} C_VEL
LIN {X 0,Y 594.258,Z 417.979,A -85,B 0,C 180,E1 -1263.39,E2 -1263.39} C_VEL
LIN {X 0,Y 594.232,Z 414.531,A -85,B 0,C 180,E1 -1264.749,E2 -1264.749} C_VEL
LIN {X 0,Y 594.279,Z 409.787,A -85,B 0,C 180,E1 -1266.11,E2 -1266.11} C_VEL
LIN {X 0,Y 594.288,Z 403.656,A -85,B 0,C 180,E1 -1267.475,E2 -1267.475} C_VEL
LIN {X 0,Y 594.332,Z 395.932,A -85,B 0,C 180,E1 -1268.843,E2 -1268.843} C_VEL
LIN {X 0,Y 594.387,Z 387.684,A -85,B 0,C 180,E1 -1270.044,E2 -1270.044} C_VEL
LIN {X 0,Y 594.41,Z 377.98,A -85,B 0,C 180,E1 -1271.229,E2 -1271.229} C_VEL
LIN {X 0,Y 594.516,Z 367.636,A -85,B 0,C 180,E1 -1272.286,E2 -1272.286} C_VEL
LIN {X 0,Y 594.578,Z 355.575,A -85,B 0,C 180,E1 -1273.326,E2 -1273.326} C_VEL
LIN {X 0,Y 594.595,Z 352.406,A -85,B 0,C 180,E1 -1273.566,E2 -1273.566} C_VEL
LIN {X 0,Y 593.958,Z 347.82,A -85,B 0,C 180,E1 -1273.918,E2 -1273.918} C_VEL
LIN {X 0,Y 591.208,Z 340.308,A -85,B 0,C 180,E1 -1274.49,E2 -1274.49} C_VEL
LIN {X 0,Y 588.486,Z 332.527,A -85,B 0,C 180,E1 -1275.023,E2 -1275.023} C_VEL
LIN {X 0,Y 587.886,Z 327.458,A -85,B 0,C 180,E1 -1275.312,E2 -1275.312} C_VEL
LIN {X 0,Y 588.042,Z 313.783,A -85,B 0,C 180,E1 -1275.955,E2 -1275.955} C_VEL
LIN {X 0,Y 588.164,Z 298.469,A -85,B 0,C 180,E1 -1276.509,E2 -1276.509} C_VEL
LIN {X 0,Y 588.253,Z 284.643,A -85,B 0,C 180,E1 -1276.879,E2 -1276.879} C_VEL
LIN {X 0,Y 588.311,Z 268.365,A -85,B 0,C 180,E1 -1277.165,E2 -1277.165} C_VEL
LIN {X 0,Y 588.56,Z 116.398,A -85,B 0,C 180,E1 -1279.069,E2 -1279.069} C_VEL
LIN {X 0,Y 587.619,Z 111.349,A -85,B 0,C 180,E1 -1279.186,E2 -1279.186} C_VEL
LIN {X 0,Y 587.659,Z 100.035,A -85,B 0,C 180,E1 -1280.842,E2 -1280.842} C_VEL
LIN {X 0,Y 587.322,Z 97.951,A -85,B 0,C 180,E1 -1281.162,E2 -1281.162} C_VEL
LIN {X 0,Y 587.3,Z 97.956,A -85,B 0,C 180,E1 -1284.008,E2 -1284.008} C_VEL
LIN {X 0,Y 587.307,Z 97.95,A -85,B 0,C 180,E1 -1286.28,E2 -1286.28} C_VEL
LIN {X 0,Y 587.343,Z 97.944,A -85,B 0,C 180,E1 -1289.132,E2 -1289.132} C_VEL
LIN {X 0,Y 587.316,Z 97.953,A -85,B 0,C 180,E1 -1291.831,E2 -1291.831} C_VEL
LIN {X 0,Y 587.331,Z 97.945,A -85,B 0,C 180,E1 -1294.345,E2 -1294.345} C_VEL
LIN {X 0,Y 587.34,Z 97.951,A -85,B 0,C 180,E1 -1297.608,E2 -1297.608} C_VEL
LIN {X 0,Y 587.306,Z 97.947,A -85,B 0,C 180,E1 -1300.255,E2 -1300.255} C_VEL
LIN {X 0,Y 587.292,Z 97.955,A -85,B 0,C 180,E1 -1303.116,E2 -1303.116} C_VEL
LIN {X 0,Y 587.3,Z 97.946,A -85,B 0,C 180,E1 -1306.047,E2 -1306.047} C_VEL
LIN {X 0,Y 587.333,Z 97.948,A -85,B 0,C 180,E1 -1308.926,E2 -1308.926} C_VEL
LIN {X 0,Y 587.315,Z 97.95,A -85,B 0,C 180,E1 -1311.519,E2 -1311.519} C_VEL
LIN {X 0,Y 587.278,Z 97.948,A -85,B 0,C 180,E1 -1314.099,E2 -1314.099} C_VEL
LIN {X 0,Y 587.334,Z 97.951,A -85,B 0,C 180,E1 -1316.89,E2 -1316.89} C_VEL
LIN {X 0,Y 587.296,Z 97.947,A -85,B 0,C 180,E1 -1319.828,E2 -1319.828} C_VEL
LIN {X 0,Y 587.299,Z 97.95,A -85,B 0,C 180,E1 -1322.318,E2 -1322.318} C_VEL
LIN {X 0,Y 587.3,Z 97.95,A -85,B 0,C 180,E1 -1325.239,E2 -1325.239} C_VEL
LIN {X 0,Y 587.3,Z 97.951,A -85,B 0,C 180,E1 -1328.225,E2 -1328.225} C_VEL
LIN {X 0,Y 587.324,Z 97.947,A -85,B 0,C 180,E1 -1331.15,E2 -1331.15} C_VEL
LIN {X 0,Y 587.288,Z 97.951,A -85,B 0,C 180,E1 -1334.024,E2 -1334.024} C_VEL
LIN {X 0,Y 587.324,Z 97.95,A -85,B 0,C 180,E1 -1336.153,E2 -1336.153} C_VEL
LIN {X 0,Y 587.342,Z 97.945,A -85,B 0,C 180,E1 -1338.962,E2 -1338.962} C_VEL
LIN {X 0,Y 587.328,Z 97.946,A -85,B 0,C 180,E1 -1341.744,E2 -1341.744} C_VEL
LIN {X 0,Y 587.334,Z 97.95,A -85,B 0,C 180,E1 -1344.507,E2 -1344.507} C_VEL
LIN {X 0,Y 587.333,Z 97.945,A -85,B 0,C 180,E1 -1347.257,E2 -1347.257} C_VEL
LIN {X 0,Y 587.382,Z 97.947,A -85,B 0,C 180,E1 -1350,E2 -1350} C_VEL
LIN {X 0,Y 587.343,Z 98.027,A -85,B 0,C 180,E1 -1352.529,E2 -1352.529} C_VEL
LIN {X 0,Y 588.061,Z 103.44,A -85,B 0,C 180,E1 -1353.254,E2 -1353.254} C_VEL
LIN {X 0,Y 587.813,Z 126.495,A -85,B 0,C 180,E1 -1356.177,E2 -1356.177} C_VEL
LIN {X 0,Y 587.739,Z 140.383,A -85,B 0,C 180,E1 -1357.914,E2 -1357.914} C_VEL
LIN {X 0,Y 588.569,Z 145.171,A -85,B 0,C 180,E1 -1358.006,E2 -1358.006} C_VEL
LIN {X 0,Y 588.294,Z 306.107,A -85,B 0,C 180,E1 -1360.04,E2 -1360.04} C_VEL
LIN {X 0,Y 588.181,Z 321.095,A -85,B 0,C 180,E1 -1360.368,E2 -1360.368} C_VEL
LIN {X 0,Y 588.099,Z 335.211,A -85,B 0,C 180,E1 -1360.805,E2 -1360.805} C_VEL
LIN {X 0,Y 587.994,Z 350.795,A -85,B 0,C 180,E1 -1361.446,E2 -1361.446} C_VEL
LIN {X 0,Y 587.834,Z 364.444,A -85,B 0,C 180,E1 -1362.165,E2 -1362.165} C_VEL
LIN {X 0,Y 587.702,Z 376.87,A -85,B 0,C 180,E1 -1362.957,E2 -1362.957} C_VEL
LIN {X 0,Y 587.584,Z 389.763,A -85,B 0,C 180,E1 -1363.947,E2 -1363.947} C_VEL
LIN {X 0,Y 587.472,Z 400.184,A -85,B 0,C 180,E1 -1364.904,E2 -1364.904} C_VEL
LIN {X 0,Y 587.386,Z 410.081,A -85,B 0,C 180,E1 -1365.973,E2 -1365.973} C_VEL
LIN {X 0,Y 587.312,Z 419.896,A -85,B 0,C 180,E1 -1367.231,E2 -1367.231} C_VEL
LIN {X 0,Y 587.25,Z 428.02,A -85,B 0,C 180,E1 -1368.49,E2 -1368.49} C_VEL
LIN {X 0,Y 587.227,Z 433.906,A -85,B 0,C 180,E1 -1369.579,E2 -1369.579} C_VEL
LIN {X 0,Y 587.184,Z 438.757,A -85,B 0,C 180,E1 -1370.654,E2 -1370.654} C_VEL
LIN {X 0,Y 587.173,Z 442.945,A -85,B 0,C 180,E1 -1371.78,E2 -1371.78} C_VEL
LIN {X 0,Y 587.134,Z 446.025,A -85,B 0,C 180,E1 -1372.825,E2 -1372.825} C_VEL
LIN {X 0,Y 587.116,Z 448.696,A -85,B 0,C 180,E1 -1374.016,E2 -1374.016} C_VEL
LIN {X 0,Y 587.104,Z 449.935,A -85,B 0,C 180,E1 -1374.77,E2 -1374.77} C_VEL
LIN {X 0,Y 587.128,Z 451.305,A -85,B 0,C 180,E1 -1376.289,E2 -1376.289} C_VEL
LIN {X 0,Y 587.157,Z 451.355,A -85,B 0,C 180,E1 -1377.656,E2 -1377.656} C_VEL
LIN {X 0,Y 587.164,Z 450.193,A -85,B 0,C 180,E1 -1379.1,E2 -1379.1} C_VEL
LIN {X 0,Y 587.157,Z 447.892,A -85,B 0,C 180,E1 -1380.479,E2 -1380.479} C_VEL
LIN {X 0,Y 587.141,Z 444.533,A -85,B 0,C 180,E1 -1381.803,E2 -1381.803} C_VEL
LIN {X 0,Y 587.169,Z 440.167,A -85,B 0,C 180,E1 -1383.085,E2 -1383.085} C_VEL
LIN {X 0,Y 587.187,Z 434.8,A -85,B 0,C 180,E1 -1384.324,E2 -1384.324} C_VEL
LIN {X 0,Y 587.241,Z 427.495,A -85,B 0,C 180,E1 -1385.69,E2 -1385.69} C_VEL
LIN {X 0,Y 587.3,Z 419.148,A -85,B 0,C 180,E1 -1386.965,E2 -1386.965} C_VEL
LIN {X 0,Y 587.377,Z 409.976,A -85,B 0,C 180,E1 -1388.129,E2 -1388.129} C_VEL
LIN {X 0,Y 587.487,Z 399.689,A -85,B 0,C 180,E1 -1389.234,E2 -1389.234} C_VEL
LIN {X 0,Y 587.605,Z 387.35,A -85,B 0,C 180,E1 -1390.343,E2 -1390.343} C_VEL
LIN {X 0,Y 587.715,Z 375.333,A -85,B 0,C 180,E1 -1391.239,E2 -1391.239} C_VEL
LIN {X 0,Y 587.827,Z 362.635,A -85,B 0,C 180,E1 -1392.031,E2 -1392.031} C_VEL
LIN {X 0,Y 587.982,Z 347.795,A -85,B 0,C 180,E1 -1392.782,E2 -1392.782} C_VEL
LIN {X 0,Y 588.089,Z 332.919,A -85,B 0,C 180,E1 -1393.364,E2 -1393.364} C_VEL
LIN {X 0,Y 588.233,Z 318.118,A -85,B 0,C 180,E1 -1393.798,E2 -1393.798} C_VEL
LIN {X 0,Y 588.277,Z 302.675,A -85,B 0,C 180,E1 -1394.104,E2 -1394.104} C_VEL
LIN {X 0,Y 588.478,Z 141.701,A -85,B 0,C 180,E1 -1396.131,E2 -1396.131} C_VEL
LIN {X 0,Y 587.943,Z 138.514,A -85,B 0,C 180,E1 -1396.206,E2 -1396.206} C_VEL
LIN {X 0,Y 588.208,Z 107.474,A -85,B 0,C 180,E1 -1399.257,E2 -1399.257} C_VEL
LIN {X 0,Y 588.06,Z 101.13,A -85,B 0,C 180,E1 -1399.896,E2 -1399.896} C_VEL
LIN {X 0,Y 587.335,Z 97.953,A -85,B 0,C 180,E1 -1400.265,E2 -1400.265} C_VEL
LIN {X 0,Y 587.322,Z 97.947,A -85,B 0,C 180,E1 -1403.251,E2 -1403.251} C_VEL
LIN {X 0,Y 587.359,Z 97.947,A -85,B 0,C 180,E1 -1405.779,E2 -1405.779} C_VEL
LIN {X 0,Y 587.342,Z 97.947,A -85,B 0,C 180,E1 -1408.231,E2 -1408.231} C_VEL
LIN {X 0,Y 587.353,Z 97.942,A -85,B 0,C 180,E1 -1410.866,E2 -1410.866} C_VEL
LIN {X 0,Y 587.36,Z 97.946,A -85,B 0,C 180,E1 -1413.819,E2 -1413.819} C_VEL
LIN {X 0,Y 587.326,Z 97.947,A -85,B 0,C 180,E1 -1415.993,E2 -1415.993} C_VEL
LIN {X 0,Y 587.318,Z 97.949,A -85,B 0,C 180,E1 -1418.225,E2 -1418.225} C_VEL
LIN {X 0,Y 587.379,Z 98.14,A -85,B 0,C 180,E1 -1419.56,E2 -1419.56} C_VEL
LIN {X 0,Y 587.887,Z 102.503,A -85,B 0,C 180,E1 -1420.08,E2 -1420.08} C_VEL
LIN {X 0,Y 587.808,Z 109.791,A -85,B 0,C 180,E1 -1420.911,E2 -1420.911} C_VEL
LIN {X 0,Y 588.591,Z 115.233,A -85,B 0,C 180,E1 -1421.008,E2 -1421.008} C_VEL
LIN {X 0,Y 588.278,Z 275.592,A -85,B 0,C 180,E1 -1423.035,E2 -1423.035} C_VEL
LIN {X 0,Y 588.227,Z 290.811,A -85,B 0,C 180,E1 -1423.359,E2 -1423.359} C_VEL
LIN {X 0,Y 588.088,Z 305.76,A -85,B 0,C 180,E1 -1423.823,E2 -1423.823} C_VEL
LIN {X 0,Y 587.977,Z 319.703,A -85,B 0,C 180,E1 -1424.399,E2 -1424.399} C_VEL
LIN {X 0,Y 587.833,Z 331.858,A -85,B 0,C 180,E1 -1425.016,E2 -1425.016} C_VEL
LIN {X 0,Y 587.738,Z 345.227,A -85,B 0,C 180,E1 -1425.842,E2 -1425.842} C_VEL
LIN {X 0,Y 587.581,Z 358.741,A -85,B 0,C 180,E1 -1426.864,E2 -1426.864} C_VEL
LIN {X 0,Y 587.455,Z 370.271,A -85,B 0,C 180,E1 -1427.915,E2 -1427.915} C_VEL
LIN {X 0,Y 587.349,Z 380.018,A -85,B 0,C 180,E1 -1428.962,E2 -1428.962} C_VEL
LIN {X 0,Y 587.31,Z 389.547,A -85,B 0,C 180,E1 -1430.182,E2 -1430.182} C_VEL
LIN {X 0,Y 587.268,Z 397.451,A -85,B 0,C 180,E1 -1431.397,E2 -1431.397} C_VEL
LIN {X 0,Y 587.216,Z 404.884,A -85,B 0,C 180,E1 -1432.78,E2 -1432.78} C_VEL
LIN {X 0,Y 587.227,Z 410.775,A -85,B 0,C 180,E1 -1434.161,E2 -1434.161} C_VEL
LIN {X 0,Y 587.134,Z 414.252,A -85,B 0,C 180,E1 -1435.193,E2 -1435.193} C_VEL
LIN {X 0,Y 587.179,Z 417.803,A -85,B 0,C 180,E1 -1436.569,E2 -1436.569} C_VEL
LIN {X 0,Y 587.14,Z 420.133,A -85,B 0,C 180,E1 -1437.942,E2 -1437.942} C_VEL
LIN {X 0,Y 587.135,Z 421.311,A -85,B 0,C 180,E1 -1439.314,E2 -1439.314} C_VEL
LIN {X 0,Y 587.136,Z 421.343,A -85,B 0,C 180,E1 -1440.686,E2 -1440.686} C_VEL
LIN {X 0,Y 587.14,Z 420.238,A -85,B 0,C 180,E1 -1442.058,E2 -1442.058} C_VEL
LIN {X 0,Y 587.181,Z 417.992,A -85,B 0,C 180,E1 -1443.431,E2 -1443.431} C_VEL
LIN {X 0,Y 587.134,Z 414.529,A -85,B 0,C 180,E1 -1444.806,E2 -1444.806} C_VEL
LIN {X 0,Y 587.183,Z 409.773,A -85,B 0,C 180,E1 -1446.184,E2 -1446.184} C_VEL
LIN {X 0,Y 587.216,Z 405.306,A -85,B 0,C 180,E1 -1447.219,E2 -1447.219} C_VEL
LIN {X 0,Y 587.253,Z 397.981,A -85,B 0,C 180,E1 -1448.603,E2 -1448.603} C_VEL
LIN {X 0,Y 587.305,Z 390.191,A -85,B 0,C 180,E1 -1449.818,E2 -1449.818} C_VEL
LIN {X 0,Y 587.385,Z 379.817,A -85,B 0,C 180,E1 -1451.15,E2 -1451.15} C_VEL
LIN {X 0,Y 587.492,Z 369.405,A -85,B 0,C 180,E1 -1452.259,E2 -1452.259} C_VEL
LIN {X 0,Y 587.614,Z 357.714,A -85,B 0,C 180,E1 -1453.311,E2 -1453.311} C_VEL
LIN {X 0,Y 587.765,Z 344.464,A -85,B 0,C 180,E1 -1454.3,E2 -1454.3} C_VEL
LIN {X 0,Y 587.82,Z 331.885,A -85,B 0,C 180,E1 -1455.072,E2 -1455.072} C_VEL
LIN {X 0,Y 587.986,Z 319.738,A -85,B 0,C 180,E1 -1455.69,E2 -1455.69} C_VEL
LIN {X 0,Y 588.095,Z 305.798,A -85,B 0,C 180,E1 -1456.265,E2 -1456.265} C_VEL
LIN {X 0,Y 588.232,Z 289.895,A -85,B 0,C 180,E1 -1456.753,E2 -1456.753} C_VEL
LIN {X 0,Y 588.273,Z 275.855,A -85,B 0,C 180,E1 -1457.051,E2 -1457.051} C_VEL
LIN {X 0,Y 588.496,Z 172.785,A -85,B 0,C 180,E1 -1458.359,E2 -1458.359} C_VEL
LIN {X 0,Y 588.437,Z 115.371,A -85,B 0,C 180,E1 -1459.086,E2 -1459.086} C_VEL
LIN {X 0,Y 587.615,Z 111.36,A -85,B 0,C 180,E1 -1459.185,E2 -1459.185} C_VEL
LIN {X 0,Y 587.67,Z 100.038,A -85,B 0,C 180,E1 -1460.841,E2 -1460.841} C_VEL
LIN {X 0,Y 587.335,Z 97.95,A -85,B 0,C 180,E1 -1461.182,E2 -1461.182} C_VEL
LIN {X 0,Y 587.299,Z 97.957,A -85,B 0,C 180,E1 -1464.008,E2 -1464.008} C_VEL
LIN {X 0,Y 587.306,Z 97.951,A -85,B 0,C 180,E1 -1466.28,E2 -1466.28} C_VEL
LIN {X 0,Y 587.341,Z 97.946,A -85,B 0,C 180,E1 -1469.132,E2 -1469.132} C_VEL
LIN {X 0,Y 587.314,Z 97.953,A -85,B 0,C 180,E1 -1471.831,E2 -1471.831} C_VEL
LIN {X 0,Y 587.329,Z 97.945,A -85,B 0,C 180,E1 -1474.345,E2 -1474.345} C_VEL
LIN {X 0,Y 587.337,Z 97.951,A -85,B 0,C 180,E1 -1477.608,E2 -1477.608} C_VEL
LIN {X 0,Y 587.302,Z 97.948,A -85,B 0,C 180,E1 -1480.255,E2 -1480.255} C_VEL
LIN {X 0,Y 587.289,Z 97.957,A -85,B 0,C 180,E1 -1483.115,E2 -1483.115} C_VEL
LIN {X 0,Y 587.296,Z 97.949,A -85,B 0,C 180,E1 -1486.047,E2 -1486.047} C_VEL
LIN {X 0,Y 587.33,Z 97.952,A -85,B 0,C 180,E1 -1488.926,E2 -1488.926} C_VEL
LIN {X 0,Y 587.31,Z 97.95,A -85,B 0,C 180,E1 -1491.519,E2 -1491.519} C_VEL
LIN {X 0,Y 587.263,Z 97.954,A -85,B 0,C 180,E1 -1494.098,E2 -1494.098} C_VEL
LIN {X 0,Y 587.329,Z 97.954,A -85,B 0,C 180,E1 -1496.89,E2 -1496.89} C_VEL
LIN {X 0,Y 587.29,Z 97.951,A -85,B 0,C 180,E1 -1499.827,E2 -1499.827} C_VEL
LIN {X 0,Y 587.362,Z 98.118,A -85,B 0,C 180,E1 -1502.955,E2 -1502.955} C_VEL
LIN {X 0,Y 588.33,Z 103.848,A -85,B 0,C 180,E1 -1503.627,E2 -1503.627} C_VEL
LIN {X 0,Y 588.257,Z 125.6,A -85,B 0,C 180,E1 -1506.033,E2 -1506.033} C_VEL
LIN {X 0,Y 587.995,Z 152.258,A -85,B 0,C 180,E1 -1508.987,E2 -1508.987} C_VEL
LIN {X 0,Y 587.813,Z 169.391,A -85,B 0,C 180,E1 -1510.856,E2 -1510.856} C_VEL
LIN {X 0,Y 588.62,Z 173.952,A -85,B 0,C 180,E1 -1510.947,E2 -1510.947} C_VEL
LIN {X 0,Y 588.3,Z 336.361,A -85,B 0,C 180,E1 -1512.999,E2 -1512.999} C_VEL
LIN {X 0,Y 588.217,Z 351.706,A -85,B 0,C 180,E1 -1513.336,E2 -1513.336} C_VEL
LIN {X 0,Y 588.083,Z 367.042,A -85,B 0,C 180,E1 -1513.823,E2 -1513.823} C_VEL
LIN {X 0,Y 587.997,Z 380.767,A -85,B 0,C 180,E1 -1514.399,E2 -1514.399} C_VEL
LIN {X 0,Y 587.828,Z 394.24,A -85,B 0,C 180,E1 -1515.105,E2 -1515.105} C_VEL
LIN {X 0,Y 587.741,Z 407.115,A -85,B 0,C 180,E1 -1515.929,E2 -1515.929} C_VEL
LIN {X 0,Y 587.582,Z 419.288,A -85,B 0,C 180,E1 -1516.864,E2 -1516.864} C_VEL
LIN {X 0,Y 587.454,Z 430.748,A -85,B 0,C 180,E1 -1517.915,E2 -1517.915} C_VEL
LIN {X 0,Y 587.348,Z 440.39,A -85,B 0,C 180,E1 -1518.963,E2 -1518.963} C_VEL
LIN {X 0,Y 587.305,Z 449.857,A -85,B 0,C 180,E1 -1520.182,E2 -1520.182} C_VEL
LIN {X 0,Y 587.265,Z 457.732,A -85,B 0,C 180,E1 -1521.397,E2 -1521.397} C_VEL
LIN {X 0,Y 587.215,Z 465.089,A -85,B 0,C 180,E1 -1522.781,E2 -1522.781} C_VEL
LIN {X 0,Y 587.227,Z 470.924,A -85,B 0,C 180,E1 -1524.161,E2 -1524.161} C_VEL
LIN {X 0,Y 587.136,Z 474.384,A -85,B 0,C 180,E1 -1525.194,E2 -1525.194} C_VEL
LIN {X 0,Y 587.18,Z 477.888,A -85,B 0,C 180,E1 -1526.569,E2 -1526.569} C_VEL
LIN {X 0,Y 587.14,Z 480.193,A -85,B 0,C 180,E1 -1527.942,E2 -1527.942} C_VEL
LIN {X 0,Y 587.135,Z 481.35,A -85,B 0,C 180,E1 -1529.314,E2 -1529.314} C_VEL
LIN {X 0,Y 587.135,Z 481.349,A -85,B 0,C 180,E1 -1530.686,E2 -1530.686} C_VEL
LIN {X 0,Y 587.14,Z 480.192,A -85,B 0,C 180,E1 -1532.058,E2 -1532.058} C_VEL
LIN {X 0,Y 587.18,Z 477.886,A -85,B 0,C 180,E1 -1533.431,E2 -1533.431} C_VEL
LIN {X 0,Y 587.136,Z 474.384,A -85,B 0,C 180,E1 -1534.806,E2 -1534.806} C_VEL
LIN {X 0,Y 587.18,Z 469.608,A -85,B 0,C 180,E1 -1536.184,E2 -1536.184} C_VEL
LIN {X 0,Y 587.23,Z 463.424,A -85,B 0,C 180,E1 -1537.565,E2 -1537.565} C_VEL
LIN {X 0,Y 587.266,Z 455.65,A -85,B 0,C 180,E1 -1538.95,E2 -1538.95} C_VEL
LIN {X 0,Y 587.351,Z 447.369,A -85,B 0,C 180,E1 -1540.166,E2 -1540.166} C_VEL
LIN {X 0,Y 587.4,Z 437.394,A -85,B 0,C 180,E1 -1541.386,E2 -1541.386} C_VEL
LIN {X 0,Y 587.522,Z 427.19,A -85,B 0,C 180,E1 -1542.434,E2 -1542.434} C_VEL
LIN {X 0,Y 587.629,Z 415.018,A -85,B 0,C 180,E1 -1543.487,E2 -1543.487} C_VEL
LIN {X 0,Y 587.774,Z 402.057,A -85,B 0,C 180,E1 -1544.416,E2 -1544.416} C_VEL
LIN {X 0,Y 587.89,Z 387.867,A -85,B 0,C 180,E1 -1545.248,E2 -1545.248} C_VEL
LIN {X 0,Y 588.058,Z 373.796,A -85,B 0,C 180,E1 -1545.91,E2 -1545.91} C_VEL
LIN {X 0,Y 588.164,Z 359.302,A -85,B 0,C 180,E1 -1546.442,E2 -1546.442} C_VEL
LIN {X 0,Y 588.257,Z 343.552,A -85,B 0,C 180,E1 -1546.861,E2 -1546.861} C_VEL
LIN {X 0,Y 588.296,Z 327.709,A -85,B 0,C 180,E1 -1547.129,E2 -1547.129} C_VEL
LIN {X 0,Y 588.513,Z 171.142,A -85,B 0,C 180,E1 -1549.092,E2 -1549.092} C_VEL
LIN {X 0,Y 587.981,Z 167.528,A -85,B 0,C 180,E1 -1549.175,E2 -1549.175} C_VEL
LIN {X 0,Y 588.216,Z 139.457,A -85,B 0,C 180,E1 -1551.579,E2 -1551.579} C_VEL
LIN {X 0,Y 588.549,Z 105.726,A -85,B 0,C 180,E1 -1554.517,E2 -1554.517} C_VEL
LIN {X 0,Y 588.468,Z 102.373,A -85,B 0,C 180,E1 -1554.817,E2 -1554.817} C_VEL
LIN {X 0,Y 587.301,Z 97.958,A -85,B 0,C 180,E1 -1555.281,E2 -1555.281} C_VEL
LIN {X 0,Y 587.287,Z 97.952,A -85,B 0,C 180,E1 -1557.821,E2 -1557.821} C_VEL
LIN {X 0,Y 587.293,Z 97.95,A -85,B 0,C 180,E1 -1560.173,E2 -1560.173} C_VEL
LIN {X 0,Y 587.323,Z 97.948,A -85,B 0,C 180,E1 -1562.58,E2 -1562.58} C_VEL
LIN {X 0,Y 587.302,Z 97.957,A -85,B 0,C 180,E1 -1565.057,E2 -1565.057} C_VEL
LIN {X 0,Y 587.324,Z 97.945,A -85,B 0,C 180,E1 -1567.837,E2 -1567.837} C_VEL
LIN {X 0,Y 587.3,Z 97.95,A -85,B 0,C 180,E1 -1570.256,E2 -1570.256} C_VEL
LIN {X 0,Y 587.29,Z 97.954,A -85,B 0,C 180,E1 -1573.116,E2 -1573.116} C_VEL
LIN {X 0,Y 587.298,Z 97.949,A -85,B 0,C 180,E1 -1576.047,E2 -1576.047} C_VEL
LIN {X 0,Y 587.332,Z 97.95,A -85,B 0,C 180,E1 -1578.926,E2 -1578.926} C_VEL
LIN {X 0,Y 587.31,Z 97.947,A -85,B 0,C 180,E1 -1581.519,E2 -1581.519} C_VEL
LIN {X 0,Y 587.276,Z 97.955,A -85,B 0,C 180,E1 -1584.099,E2 -1584.099} C_VEL
LIN {X 0,Y 587.332,Z 97.948,A -85,B 0,C 180,E1 -1586.89,E2 -1586.89} C_VEL
LIN {X 0,Y 587.316,Z 97.946,A -85,B 0,C 180,E1 -1589.494,E2 -1589.494} C_VEL
LIN {X 0,Y 587.299,Z 97.957,A -85,B 0,C 180,E1 -1592.18,E2 -1592.18} C_VEL
LIN {X 0,Y 587.328,Z 97.952,A -85,B 0,C 180,E1 -1594.483,E2 -1594.483} C_VEL
LIN {X 0,Y 587.307,Z 97.95,A -85,B 0,C 180,E1 -1597.485,E2 -1597.485} C_VEL
LIN {X 0,Y 587.361,Z 98.127,A -85,B 0,C 180,E1 -1598.955,E2 -1598.955} C_VEL
LIN {X 0,Y 587.714,Z 104.403,A -85,B 0,C 180,E1 -1599.892,E2 -1599.892} C_VEL
LIN {X 0,Y 587.606,Z 111.479,A -85,B 0,C 180,E1 -1600.922,E2 -1600.922} C_VEL
LIN {X 0,Y 588.57,Z 116.688,A -85,B 0,C 180,E1 -1601.025,E2 -1601.025} C_VEL
LIN {X 0,Y 588.279,Z 275.188,A -85,B 0,C 180,E1 -1603.027,E2 -1603.027} C_VEL
LIN {X 0,Y 588.214,Z 289.889,A -85,B 0,C 180,E1 -1603.337,E2 -1603.337} C_VEL
LIN {X 0,Y 588.09,Z 305.75,A -85,B 0,C 180,E1 -1603.824,E2 -1603.824} C_VEL
LIN {X 0,Y 587.976,Z 319.751,A -85,B 0,C 180,E1 -1604.399,E2 -1604.399} C_VEL
LIN {X 0,Y 587.834,Z 333.47,A -85,B 0,C 180,E1 -1605.105,E2 -1605.105} C_VEL
LIN {X 0,Y 587.747,Z 346.487,A -85,B 0,C 180,E1 -1605.932,E2 -1605.932} C_VEL
LIN {X 0,Y 587.565,Z 359.817,A -85,B 0,C 180,E1 -1606.952,E2 -1606.952} C_VEL
LIN {X 0,Y 587.472,Z 372.066,A -85,B 0,C 180,E1 -1608.091,E2 -1608.091} C_VEL
LIN {X 0,Y 587.383,Z 382.924,A -85,B 0,C 180,E1 -1609.312,E2 -1609.312} C_VEL
LIN {X 0,Y 587.285,Z 391.995,A -85,B 0,C 180,E1 -1610.529,E2 -1610.529} C_VEL
LIN {X 0,Y 587.258,Z 399.486,A -85,B 0,C 180,E1 -1611.743,E2 -1611.743} C_VEL
LIN {X 0,Y 587.207,Z 406.499,A -85,B 0,C 180,E1 -1613.126,E2 -1613.126} C_VEL
LIN {X 0,Y 587.198,Z 412.008,A -85,B 0,C 180,E1 -1614.506,E2 -1614.506} C_VEL
LIN {X 0,Y 587.169,Z 416.181,A -85,B 0,C 180,E1 -1615.882,E2 -1615.882} C_VEL
LIN {X 0,Y 587.127,Z 419.112,A -85,B 0,C 180,E1 -1617.256,E2 -1617.256} C_VEL
LIN {X 0,Y 587.143,Z 420.874,A -85,B 0,C 180,E1 -1618.628,E2 -1618.628} C_VEL
LIN {X 0,Y 587.135,Z 421.496,A -85,B 0,C 180,E1 -1620,E2 -1620} C_VEL
LIN {X 0,Y 587.145,Z 420.953,A -85,B 0,C 180,E1 -1621.372,E2 -1621.372} C_VEL
LIN {X 0,Y 587.129,Z 419.257,A -85,B 0,C 180,E1 -1622.745,E2 -1622.745} C_VEL
LIN {X 0,Y 587.169,Z 416.414,A -85,B 0,C 180,E1 -1624.119,E2 -1624.119} C_VEL
LIN {X 0,Y 587.198,Z 412.318,A -85,B 0,C 180,E1 -1625.495,E2 -1625.495} C_VEL
LIN {X 0,Y 587.208,Z 406.918,A -85,B 0,C 180,E1 -1626.874,E2 -1626.874} C_VEL
LIN {X 0,Y 587.247,Z 399.987,A -85,B 0,C 180,E1 -1628.257,E2 -1628.257} C_VEL
LIN {X 0,Y 587.287,Z 391.41,A -85,B 0,C 180,E1 -1629.645,E2 -1629.645} C_VEL
LIN {X 0,Y 587.346,Z 382.233,A -85,B 0,C 180,E1 -1630.863,E2 -1630.863} C_VEL
LIN {X 0,Y 587.447,Z 372.928,A -85,B 0,C 180,E1 -1631.91,E2 -1631.91} C_VEL
LIN {X 0,Y 587.559,Z 361.861,A -85,B 0,C 180,E1 -1632.961,E2 -1632.961} C_VEL
LIN {X 0,Y 587.711,Z 349.429,A -85,B 0,C 180,E1 -1633.953,E2 -1633.953} C_VEL
LIN {X 0,Y 587.821,Z 336.47,A -85,B 0,C 180,E1 -1634.807,E2 -1634.807} C_VEL
LIN {X 0,Y 587.886,Z 327.458,A -85,B 0,C 180,E1 -1635.312,E2 -1635.312} C_VEL
LIN {X 0,Y 587.34,Z 322.311,A -85,B 0,C 180,E1 -1635.59,E2 -1635.59} C_VEL
LIN {X 0,Y 584.732,Z 313.962,A -85,B 0,C 180,E1 -1636.045,E2 -1636.045} C_VEL
LIN {X 0,Y 582.05,Z 305.416,A -85,B 0,C 180,E1 -1636.459,E2 -1636.459} C_VEL
LIN {X 0,Y 581.334,Z 299.936,A -85,B 0,C 180,E1 -1636.662,E2 -1636.662} C_VEL
LIN {X 0,Y 581.445,Z 285.787,A -85,B 0,C 180,E1 -1637.054,E2 -1637.054} C_VEL
LIN {X 0,Y 581.528,Z 270.738,A -85,B 0,C 180,E1 -1637.339,E2 -1637.339} C_VEL
LIN {X 0,Y 581.892,Z 117.632,A -85,B 0,C 180,E1 -1639.279,E2 -1639.279} C_VEL
LIN {X 0,Y 580.664,Z 111.402,A -85,B 0,C 180,E1 -1639.417,E2 -1639.417} C_VEL
LIN {X 0,Y 580.723,Z 101.544,A -85,B 0,C 180,E1 -1640.877,E2 -1640.877} C_VEL
LIN {X 0,Y 580.284,Z 98.829,A -85,B 0,C 180,E1 -1641.306,E2 -1641.306} C_VEL
LIN {X 0,Y 580.279,Z 98.827,A -85,B 0,C 180,E1 -1644.317,E2 -1644.317} C_VEL
LIN {X 0,Y 580.255,Z 98.826,A -85,B 0,C 180,E1 -1646.625,E2 -1646.625} C_VEL
LIN {X 0,Y 580.277,Z 98.826,A -85,B 0,C 180,E1 -1649.305,E2 -1649.305} C_VEL
LIN {X 0,Y 580.285,Z 98.824,A -85,B 0,C 180,E1 -1652.202,E2 -1652.202} C_VEL
LIN {X 0,Y 580.278,Z 98.823,A -85,B 0,C 180,E1 -1654.697,E2 -1654.697} C_VEL
LIN {X 0,Y 580.287,Z 98.827,A -85,B 0,C 180,E1 -1657.27,E2 -1657.27} C_VEL
LIN {X 0,Y 580.285,Z 98.822,A -85,B 0,C 180,E1 -1660.27,E2 -1660.27} C_VEL
LIN {X 0,Y 580.255,Z 98.827,A -85,B 0,C 180,E1 -1662.709,E2 -1662.709} C_VEL
LIN {X 0,Y 580.252,Z 98.827,A -85,B 0,C 180,E1 -1665.611,E2 -1665.611} C_VEL
LIN {X 0,Y 580.271,Z 98.824,A -85,B 0,C 180,E1 -1668.67,E2 -1668.67} C_VEL
LIN {X 0,Y 580.267,Z 98.831,A -85,B 0,C 180,E1 -1670.964,E2 -1670.964} C_VEL
LIN {X 0,Y 580.246,Z 98.827,A -85,B 0,C 180,E1 -1673.595,E2 -1673.595} C_VEL
LIN {X 0,Y 580.274,Z 98.823,A -85,B 0,C 180,E1 -1676.142,E2 -1676.142} C_VEL
LIN {X 0,Y 580.254,Z 98.83,A -85,B 0,C 180,E1 -1678.613,E2 -1678.613} C_VEL
LIN {X 0,Y 580.278,Z 98.83,A -85,B 0,C 180,E1 -1681.023,E2 -1681.023} C_VEL
LIN {X 0,Y 580.263,Z 98.825,A -85,B 0,C 180,E1 -1683.673,E2 -1683.673} C_VEL
LIN {X 0,Y 580.244,Z 98.83,A -85,B 0,C 180,E1 -1686.441,E2 -1686.441} C_VEL
LIN {X 0,Y 580.253,Z 98.826,A -85,B 0,C 180,E1 -1689.436,E2 -1689.436} C_VEL
LIN {X 0,Y 580.237,Z 98.828,A -85,B 0,C 180,E1 -1691.644,E2 -1691.644} C_VEL
LIN {X 0,Y 580.267,Z 98.833,A -85,B 0,C 180,E1 -1694.546,E2 -1694.546} C_VEL
LIN {X 0,Y 580.23,Z 98.835,A -85,B 0,C 180,E1 -1696.695,E2 -1696.695} C_VEL
LIN {X 0,Y 580.31,Z 98.822,A -85,B 0,C 180,E1 -1698.827,E2 -1698.827} C_VEL
LIN {X 0,Y 580.295,Z 98.822,A -85,B 0,C 180,E1 -1701.643,E2 -1701.643} C_VEL
LIN {X 0,Y 580.302,Z 98.828,A -85,B 0,C 180,E1 -1704.44,E2 -1704.44} C_VEL
LIN {X 0,Y 580.339,Z 98.822,A -85,B 0,C 180,E1 -1707.918,E2 -1707.918} C_VEL
LIN {X 0,Y 580.35,Z 98.823,A -85,B 0,C 180,E1 -1710,E2 -1710} C_VEL
LIN {X 0,Y 580.306,Z 98.891,A -85,B 0,C 180,E1 -1712.343,E2 -1712.343} C_VEL
LIN {X 0,Y 581.191,Z 104.621,A -85,B 0,C 180,E1 -1713.119,E2 -1713.119} C_VEL
LIN {X 0,Y 580.929,Z 126.37,A -85,B 0,C 180,E1 -1715.902,E2 -1715.902} C_VEL
LIN {X 0,Y 580.856,Z 140.636,A -85,B 0,C 180,E1 -1717.685,E2 -1717.685} C_VEL
LIN {X 0,Y 581.871,Z 146.111,A -85,B 0,C 180,E1 -1717.79,E2 -1717.79} C_VEL
LIN {X 0,Y 581.505,Z 305.729,A -85,B 0,C 180,E1 -1719.829,E2 -1719.829} C_VEL
LIN {X 0,Y 581.407,Z 319.942,A -85,B 0,C 180,E1 -1720.139,E2 -1720.139} C_VEL
LIN {X 0,Y 581.316,Z 333.056,A -85,B 0,C 180,E1 -1720.536,E2 -1720.536} C_VEL
LIN {X 0,Y 581.165,Z 346.686,A -85,B 0,C 180,E1 -1721.068,E2 -1721.068} C_VEL
LIN {X 0,Y 580.955,Z 361.276,A -85,B 0,C 180,E1 -1721.8,E2 -1721.8} C_VEL
LIN {X 0,Y 580.81,Z 373.873,A -85,B 0,C 180,E1 -1722.58,E2 -1722.58} C_VEL
LIN {X 0,Y 580.671,Z 385.955,A -85,B 0,C 180,E1 -1723.473,E2 -1723.473} C_VEL
LIN {X 0,Y 580.494,Z 398.836,A -85,B 0,C 180,E1 -1724.621,E2 -1724.621} C_VEL
LIN {X 0,Y 580.374,Z 408.309,A -85,B 0,C 180,E1 -1725.631,E2 -1725.631} C_VEL
LIN {X 0,Y 580.257,Z 417.64,A -85,B 0,C 180,E1 -1726.797,E2 -1726.797} C_VEL
LIN {X 0,Y 580.215,Z 425.683,A -85,B 0,C 180,E1 -1727.991,E2 -1727.991} C_VEL
LIN {X 0,Y 580.159,Z 433.762,A -85,B 0,C 180,E1 -1729.459,E2 -1729.459} C_VEL
LIN {X 0,Y 580.095,Z 439.799,A -85,B 0,C 180,E1 -1730.839,E2 -1730.839} C_VEL
LIN {X 0,Y 580.074,Z 444.021,A -85,B 0,C 180,E1 -1732.061,E2 -1732.061} C_VEL
LIN {X 0,Y 580.024,Z 447.897,A -85,B 0,C 180,E1 -1733.569,E2 -1733.569} C_VEL
LIN {X 0,Y 580.009,Z 450.337,A -85,B 0,C 180,E1 -1735.094,E2 -1735.094} C_VEL
LIN {X 0,Y 580.047,Z 451.299,A -85,B 0,C 180,E1 -1736.284,E2 -1736.284} C_VEL
LIN {X 0,Y 580.046,Z 451.298,A -85,B 0,C 180,E1 -1737.811,E2 -1737.811} C_VEL
LIN {X 0,Y 580.07,Z 450.032,A -85,B 0,C 180,E1 -1739.268,E2 -1739.268} C_VEL
LIN {X 0,Y 580.066,Z 447.615,A -85,B 0,C 180,E1 -1740.657,E2 -1740.657} C_VEL
LIN {X 0,Y 580.081,Z 443.444,A -85,B 0,C 180,E1 -1742.214,E2 -1742.214} C_VEL
LIN {X 0,Y 580.096,Z 438.615,A -85,B 0,C 180,E1 -1743.55,E2 -1743.55} C_VEL
LIN {X 0,Y 580.167,Z 431.241,A -85,B 0,C 180,E1 -1745.128,E2 -1745.128} C_VEL
LIN {X 0,Y 580.23,Z 423.712,A -85,B 0,C 180,E1 -1746.406,E2 -1746.406} C_VEL
LIN {X 0,Y 580.293,Z 416.192,A -85,B 0,C 180,E1 -1747.487,E2 -1747.487} C_VEL
LIN {X 0,Y 580.37,Z 407.262,A -85,B 0,C 180,E1 -1748.582,E2 -1748.582} C_VEL
LIN {X 0,Y 580.542,Z 395.203,A -85,B 0,C 180,E1 -1749.815,E2 -1749.815} C_VEL
LIN {X 0,Y 580.662,Z 385.31,A -85,B 0,C 180,E1 -1750.668,E2 -1750.668} C_VEL
LIN {X 0,Y 580.81,Z 373.786,A -85,B 0,C 180,E1 -1751.516,E2 -1751.516} C_VEL
LIN {X 0,Y 580.981,Z 361.603,A -85,B 0,C 180,E1 -1752.271,E2 -1752.271} C_VEL
LIN {X 0,Y 581.151,Z 346.258,A -85,B 0,C 180,E1 -1753.04,E2 -1753.04} C_VEL
LIN {X 0,Y 581.265,Z 332.76,A -85,B 0,C 180,E1 -1753.565,E2 -1753.565} C_VEL
LIN {X 0,Y 581.423,Z 318.669,A -85,B 0,C 180,E1 -1753.985,E2 -1753.985} C_VEL
LIN {X 0,Y 581.536,Z 303.87,A -85,B 0,C 180,E1 -1754.291,E2 -1754.291} C_VEL
LIN {X 0,Y 581.847,Z 143.054,A -85,B 0,C 180,E1 -1756.34,E2 -1756.34} C_VEL
LIN {X 0,Y 581.065,Z 138.511,A -85,B 0,C 180,E1 -1756.442,E2 -1756.442} C_VEL
LIN {X 0,Y 581.391,Z 108.042,A -85,B 0,C 180,E1 -1759.474,E2 -1759.474} C_VEL
LIN {X 0,Y 581.25,Z 102.939,A -85,B 0,C 180,E1 -1759.993,E2 -1759.993} C_VEL
LIN {X 0,Y 580.31,Z 98.828,A -85,B 0,C 180,E1 -1760.474,E2 -1760.474} C_VEL
LIN {X 0,Y 580.281,Z 98.825,A -85,B 0,C 180,E1 -1763.068,E2 -1763.068} C_VEL
LIN {X 0,Y 580.316,Z 98.826,A -85,B 0,C 180,E1 -1766.145,E2 -1766.145} C_VEL
LIN {X 0,Y 580.278,Z 98.824,A -85,B 0,C 180,E1 -1768.614,E2 -1768.614} C_VEL
LIN {X 0,Y 580.296,Z 98.822,A -85,B 0,C 180,E1 -1771.024,E2 -1771.024} C_VEL
LIN {X 0,Y 580.293,Z 98.828,A -85,B 0,C 180,E1 -1773.666,E2 -1773.666} C_VEL
LIN {X 0,Y 580.298,Z 98.826,A -85,B 0,C 180,E1 -1775.683,E2 -1775.683} C_VEL
LIN {X 0,Y 580.27,Z 98.828,A -85,B 0,C 180,E1 -1777.947,E2 -1777.947} C_VEL
LIN {X 0,Y 580.336,Z 98.984,A -85,B 0,C 180,E1 -1779.398,E2 -1779.398} C_VEL
LIN {X 0,Y 580.998,Z 102.508,A -85,B 0,C 180,E1 -1779.833,E2 -1779.833} C_VEL
LIN {X 0,Y 580.91,Z 109.819,A -85,B 0,C 180,E1 -1780.677,E2 -1780.677} C_VEL
LIN {X 0,Y 581.878,Z 115.351,A -85,B 0,C 180,E1 -1780.781,E2 -1780.781} C_VEL
LIN {X 0,Y 581.496,Z 274.678,A -85,B 0,C 180,E1 -1782.817,E2 -1782.817} C_VEL
LIN {X 0,Y 581.448,Z 288.549,A -85,B 0,C 180,E1 -1783.103,E2 -1783.103} C_VEL
LIN {X 0,Y 581.271,Z 304.571,A -85,B 0,C 180,E1 -1783.583,E2 -1783.583} C_VEL
LIN {X 0,Y 581.155,Z 317.78,A -85,B 0,C 180,E1 -1784.121,E2 -1784.121} C_VEL
LIN {X 0,Y 580.984,Z 330.237,A -85,B 0,C 180,E1 -1784.745,E2 -1784.745} C_VEL
LIN {X 0,Y 580.842,Z 342.085,A -85,B 0,C 180,E1 -1785.461,E2 -1785.461} C_VEL
LIN {X 0,Y 580.693,Z 354.422,A -85,B 0,C 180,E1 -1786.349,E2 -1786.349} C_VEL
LIN {X 0,Y 580.535,Z 366.684,A -85,B 0,C 180,E1 -1787.413,E2 -1787.413} C_VEL
